	IF NOT fbAdsReadLatchStatus.BUSY THEN
		IF fbAdsReadLatchStatus.ERR THEN
			Error := TRUE;
			ErrorID := fbAdsReadLatchStatus.ERRID;
		ELSE
			IF iTriggerInput.Edge = FallingEdge THEN
				TouchProbeActive[iTriggerInput.TouchProbe] := stTouchProbeStatusResponse.FallingEdgeActive;
				TouchProbeValid[iTriggerInput.TouchProbe] := stTouchProbeStatusResponse.FallingEdgeValid;
				TouchProbeValue[iTriggerInput.TouchProbe] := stTouchProbeStatusResponse.FallingEdgeValue;
				TouchProbeCounter[iTriggerInput.TouchProbe] := stTouchProbeStatusResponse.FallingEdgeCounter;
			ELSE
				TouchProbeActive[iTriggerInput.TouchProbe] := stTouchProbeStatusResponse.RisingEdgeActive;
				TouchProbeValid[iTriggerInput.TouchProbe] := stTouchProbeStatusResponse.RisingEdgeValid;
				TouchProbeValue[iTriggerInput.TouchProbe] := stTouchProbeStatusResponse.RisingEdgeValue;
				TouchProbeCounter[iTriggerInput.TouchProbe] := stTouchProbeStatusResponse.RisingEdgeCounter;
			END_IF
			IF TouchProbeValid[iTriggerInput.TouchProbe] = 1 THEN
				IF  iTriggerInput.Mode <> TOUCHPROBEMODE_CONTINOUS		(* single mode *)
					OR LastTouchProbeValue[ iTriggerInput.TouchProbe ] <> TouchProbeValue[ iTriggerInput.TouchProbe ] 	(* or continous mode and value changed *)
					OR LastTouchProbeCounter[ iTriggerInput.TouchProbe ] <> TouchProbeCounter[ iTriggerInput.TouchProbe ](* or continous mode and counter changed *)
					THEN (* new position recorded  *)
					RecordedPosition:=TouchProbeValue[iTriggerInput.TouchProbe];
					LastTouchProbeValue := TouchProbeValue;
					LastTouchProbeCounter := TouchProbeCounter;
					Done := TRUE;
					IF TriggerInput.ModuloPositions AND (ModuloFactor<>0) THEN	(* check for  (ModuloFactor=0) - 2007-02-06 KSt *)
						RecordedPosition := MODABS(RecordedPosition,  ModuloFactor);
						TouchProbeModuloValue[TriggerInput.TouchProbe] := RecordedPosition;
(*						InWindow := (RecordedPosition>=FirstPosition) AND (RecordedPosition<=LastPosition);*)	(* 20110216 KSt *)
						IF FirstPosition>LastPosition THEN (* 20110216 KSt *)
							InWindow := (RecordedPosition>=FirstPosition) OR  (RecordedPosition<=LastPosition);  (* 20110216 KSt *)
						ELSE
							InWindow := (RecordedPosition>=FirstPosition) AND (RecordedPosition<=LastPosition);
						END_IF
					ELSE
						InWindow := (RecordedPosition>=FirstPosition) AND (RecordedPosition<=LastPosition);
					END_IF
					IF WindowOnly AND NOT InWindow THEN
						RecordedPosition:=0;
						Done := FALSE;
						Restart := TRUE; (* ignore this event, latch next one *)
					ELSE
						(* fill RecordedData structure *)
						RecordedData.RecordedPosition := RecordedPosition;
						RecordedData.Counter:=TouchProbeCounter[TriggerInput.TouchProbe];
						RecordedData.AbsolutePosition := TouchProbeValue[iTriggerInput.TouchProbe];
						IF ModuloFactor = 0 THEN
							RecordedData.ModuloPosition := MODABS(RecordedData.AbsolutePosition,  360);
						ELSE
							RecordedData.ModuloPosition := MODABS(RecordedData.AbsolutePosition,  ModuloFactor);
						END_IF
					END_IF
					iState := STATE_INITIALIZATION;
				END_IF
			ELSIF TouchProbeActive[iTriggerInput.TouchProbe] <> 1 THEN
				TouchProbeInactiveCounter[iTriggerInput.TouchProbe] := TouchProbeInactiveCounter[iTriggerInput.TouchProbe] + 1;
				IF TouchProbeInactiveCounter[iTriggerInput.TouchProbe] > 1 THEN
					(* error condition when the probing sequence is inactive more than once *)
					Error := TRUE;
					ErrorID := MC_ERROR_TOUCH_PROBE_DEACTIVATED;
					CommandAborted := TRUE;
					iState := STATE_INITIALIZATION;
				END_IF
			END_IF
		END_IF
		fbAdsReadLatchStatus(WRTRD:=FALSE); (* reset *)
		IF iTriggerInput.Mode=TOUCHPROBEMODE_CONTINOUS AND Execute THEN
			fbAdsReadLatchStatus(WRTRD:=TRUE); (* retrigger *)
		END_IF
	END_IF
END_IF
END_ACTION

ACTION ActTouchProbeMonitorLatchValid:
(* monitor if the touch probe has been triggered *)

IF F_AxisExternalLatchValid(Axis.NcToPlc.StateDWord) THEN
	(* read the status of the latch *)
	fbAdsReadValid(	NETID:= TcMcGlobal.NCNETID_TCMC,
				PORT:=AMSPORT_R0_NCSAF ,
				IDXGRP:=16#5100+TriggerInput.EncoderID ,
				IDXOFFS:= 16#202,
				LEN:= SIZEOF(TouchProbeValid[1]),
				DESTADDR:=ADR(TouchProbeValid) ,
				READ:=TRUE ,
				TMOUT:=TcMcGlobal.tADSTimeOut );
	(* read the latched value *)
	fbAdsReadValue(	NETID:= TcMcGlobal.NCNETID_TCMC,
				PORT:=AMSPORT_R0_NCSAF ,
				IDXGRP:=16#5100+TriggerInput.EncoderID ,
				IDXOFFS:= 16#205,
				LEN:=SIZEOF(TouchProbeValue[1]),
				DESTADDR:=ADR(TouchProbeValue) ,
				READ:=TRUE ,
				TMOUT:=TcMcGlobal.tADSTimeOut );
	IF NOT fbAdsReadValid.BUSY AND NOT fbAdsReadValue.BUSY THEN
		IF fbAdsReadValid.err THEN
			Error := TRUE;
			ErrorID := fbAdsReadValid.ERRID;
			iState := STATE_INITIALIZATION;
		ELSIF fbAdsReadValue.err THEN
			Error := TRUE;
			ErrorID := fbAdsReadValue.ERRID;
			iState := STATE_INITIALIZATION;
		ELSE (* no error *)
			IF TouchProbeValid[TriggerInput.TouchProbe]=1 THEN
				RecordedPosition:=TouchProbeValue[TriggerInput.TouchProbe];
				Done := TRUE;
//				IF TriggerInput.ModuloPositions AND (ModuloFactor<>0) THEN	(* check for  (ModuloFactor=0) - 2007-02-06 KSt *)
				IF TriggerInput.ModuloPositions THEN	(* check for  (ModuloFactor=0) - 2007-02-06 KSt *)
//					RecordedPosition := MODABS(RecordedPosition,  ModuloFactor);
					IF ModuloFactor = 0 THEN (* not supposed to happen here - 2017-04-28 KSt *)
						RecordedPosition := MODABS(RecordedPosition,  360); (* default 360 not supposed to happen here - 2017-04-28 KSt *)
					ELSE
						RecordedPosition := MODABS(RecordedPosition,  ModuloFactor);
					END_IF
					TouchProbeModuloValue[TriggerInput.TouchProbe] := RecordedPosition;
(*					InWindow := (RecordedPosition>=FirstPosition) AND (RecordedPosition<=LastPosition);*)  (* 20110216 KSt *)
					IF FirstPosition>LastPosition THEN (* 20110216 KSt *)
						InWindow := (RecordedPosition>=FirstPosition) OR  (RecordedPosition<=LastPosition);  (* 20110216 KSt *)
					ELSE
						InWindow := (RecordedPosition>=FirstPosition) AND (RecordedPosition<=LastPosition);
					END_IF
				ELSE
					InWindow := (RecordedPosition>=FirstPosition) AND (RecordedPosition<=LastPosition);
				END_IF
				IF WindowOnly AND NOT InWindow THEN
					RecordedPosition:=0;
					Done := FALSE;
					Restart := TRUE; (* ignore this event, latch next one *)
				ELSE
					(* fill RecordedData structure *)
					RecordedData.RecordedPosition := RecordedPosition;
					RecordedData.Counter:=TouchProbeCounter[TriggerInput.TouchProbe];
					RecordedData.AbsolutePosition := TouchProbeValue[TriggerInput.TouchProbe];
					IF ModuloFactor = 0 THEN
						RecordedData.ModuloPosition := MODABS(RecordedData.AbsolutePosition,  360);
					ELSE
						RecordedData.ModuloPosition := MODABS(RecordedData.AbsolutePosition,  ModuloFactor);
					END_IF
				END_IF
				iState := STATE_INITIALIZATION;
			ELSE
				fbAdsReadValid(READ:=FALSE);
				fbAdsReadValue(READ:=FALSE);
			END_IF
		END_IF
	END_IF
END_IF
END_ACTION

ACTION ActTouchProbeMonitorPlcEvent:
(* touch probe sequence for simple PLC inputs *)
(* monitor PLC input trigger *)

RtrigPlcEvent(CLK:=TriggerInput.PlcEvent);
FtrigPlcEvent(CLK:=TriggerInput.PlcEvent);
IF ((TriggerInput.Edge=RisingEdge) AND RtrigPlcEvent.Q) OR
   ((TriggerInput.Edge=FallingEdge) AND FtrigPlcEvent.Q) THEN
	RecordedPosition:=Axis.NcToPlc.ActPos; 	(* 2007-02-06 KSt *)
	IF TriggerInput.ModuloPositions AND (ModuloFactor<>0) THEN	(* check for  (ModuloFactor=0) - 2007-02-06 KSt *)
		RecordedPosition :=  MODABS(RecordedPosition,  ModuloFactor);
(*		InWindow := (RecordedPosition>=FirstPosition) AND (RecordedPosition<=LastPosition);*)  (* 20110216 KSt *)
		IF FirstPosition>LastPosition THEN (* 20110216 KSt *)
			InWindow := (RecordedPosition>=FirstPosition) OR  (RecordedPosition<=LastPosition);  (* 20110216 KSt *)
		ELSE
			InWindow := (RecordedPosition>=FirstPosition) AND (RecordedPosition<=LastPosition);
		END_IF
	ELSE
		InWindow := (RecordedPosition>=FirstPosition) AND (RecordedPosition<=LastPosition);
	END_IF
	IF WindowOnly AND NOT InWindow THEN
		RecordedPosition:=0;	(* 2007-02-06 KSt *)
	ELSE
		(* fill RecordedData structure *)
		RecordedData.RecordedPosition := RecordedPosition;
		RecordedData.Counter := RecordedData.Counter + 1;
		RecordedData.AbsolutePosition := Axis.NcToPlc.ActPos;
		IF ModuloFactor = 0 THEN
			RecordedData.ModuloPosition := MODABS(RecordedData.AbsolutePosition,  360);
		ELSE
			RecordedData.ModuloPosition := MODABS(RecordedData.AbsolutePosition,  ModuloFactor);
		END_IF
		Done := TRUE;
		iState := STATE_INITIALIZATION;
	END_IF
END_IF
END_ACTION

ACTION ActTouchProbeStartupInit:
(* initialization on plc start-up *)
(* read the axis' modulo factor *)

IF TriggerInput.ModuloPositions THEN
	IF ModuloFactor = 0 THEN
		InitDone := FALSE; (* 2007-02-06 KSt *)
	END_IF
	fbAdsReadModulo(	NETID:= TcMcGlobal.NCNETID_TCMC,
						PORT:= AMSPORT_R0_NCSAF,
						IDXGRP:= 16#5000+TriggerInput.EncoderID ,
						IDXOFFS:= 16#9,
						LEN:= SIZEOF(tempModuloFactor), (* ModuloFactor changed to tempModuloFactor - 2017-40-28 KSt *)
						DESTADDR:= ADR(tempModuloFactor),
						READ:= TRUE,
						TMOUT:= TcMcGlobal.tADSTimeOut);
	IF NOT fbAdsReadModulo.BUSY THEN
		IF fbAdsReadModulo.ERR OR (tempModuloFactor=0) THEN
			fbAdsReadModulo( READ:=FALSE ); 	(* 2007-02-06 KSt *)
			InitDone := FALSE; 	(* init failed - 2007-02-06 KSt *)
			Error := TRUE;
			ErrorID := fbAdsReadModulo.ERRID;
		ELSE
			ModuloFactor := tempModuloFactor; (* take as valid ModuloFactor - 2017-04-28 KSt *) 
			InitDone := TRUE;
		END_IF
	END_IF
ELSE (* no modulo positions *)
	fbAdsReadModulo( READ:=FALSE );	(* 2007-02-06 KSt *)
	InitDone := TRUE;
END_IF
END_ACTION

END_FUNCTION_BLOCK

// POUs/Administrative/Touch Probe/MC_AbortTrigger
FUNCTION_BLOCK MC_AbortTrigger
(*	The function block is used to abort function blocks which are connected to
	trigger events (e.g. MC_TouchProbe) 
*)
VAR_IN_OUT
	Axis			:	AXIS_REF; (*Reference to an axis*)
	TriggerInput	: 	TRIGGER_REF; 		(* Reference to the trigger signal source. *)
END_VAR
VAR_INPUT
	Execute		:	BOOL;		(* Starts aborting  touch probe sequence *)
END_VAR
VAR_OUTPUT
	Done		:	BOOL;		(* function completed *)
	Busy		: 	BOOL;		(* function block is currently Busy *)
	Error		:	BOOL;		(* Signals that error has occurred within Function Block *)
{attribute 'displaymode':='hex'}
	ErrorID		:	UDINT;		(* Error identification *)
END_VAR
VAR
	ADSbusy	: 	BOOL;
	fbADSwrite	: 	ADSWRITE;
	i: INT;
	iState		: 	_E_TcMC_STATES := STATE_INITIALIZATION;
END_VAR
VAR
	LatchID		: 	UDINT;
	fbOnTrigger	: 	R_TRIG;
	stTouchProbeDeactivation : _ST_TcNc_TouchProbeDeactivation;
END_VAR

IF NOT Execute THEN
	Done := FALSE;
	Error := FALSE;			(* reset at falling edge of Execute *)
	ErrorID := 0;
END_IF

fbOnTrigger(CLK:= Execute);

FOR i := 1 TO 2 DO (* typically aborted after one scan *)
	CASE iState OF
		STATE_INITIALIZATION :

			IF fbOnTrigger.Q OR fbADSwrite.BUSY THEN
				Busy := TRUE;

				IF fbOnTrigger.Q THEN
					(* initialization *)
					Done := FALSE;
					Error := FALSE;
					ErrorID := 0;
					fbADSwrite(WRITE:=FALSE);
					IF TriggerInput.EncoderID > 255 THEN
						Error := TRUE;
						ErrorID := MC_ERROR_INVALID_TOUCH_PROBE;
					END_IF
				END_IF

				IF TcMcGlobal.NcDeviceInfoNcVersion=0 THEN
					(* read version of NC *)
					TcMcGlobal.ReadDeviceInfo();
					iState := STATE_WAITING;
					EXIT; (* FOR loop *)
				ELSIF NOT Error THEN
					iState := STATE_ORDER;
				END_IF
			END_IF

		STATE_WAITING :	(* 2013-09-04 - new waiting state in case of invalid NC version information *)
			(* check for NC version *)
			TcMcGlobal.ReadDeviceInfo();
			IF NOT TcMcGlobal.fbADSRDDEVINFO.BUSY THEN
				istate := STATE_ORDER;
			ELSE
				EXIT; (* FOR loop *)
			END_IF

		STATE_ORDER :
			CASE TriggerInput.TouchProbe OF
				TouchProbe1,
				TouchProbe2,
				TouchProbe3,
				TouchProbe4:
					IF TcMcGlobal.NcDeviceInfoNcVersion > 16#020B07DD AND (TriggerInput.mode<>TOUCHPROBEMODE_SINGLE_COMPATIBILITYMODE) THEN
						(* new touch probe interface since TwinCAT 2.11 Nc-Driver 2014 *)
						stTouchProbeDeactivation.TouchProbe := TriggerInput.TouchProbe;
						stTouchProbeDeactivation.Edge := TriggerInput.Edge;
						fbADSwrite(	NETID:= TcMcGlobal.NCNETID_TCMC,
									PORT:=AMSPORT_R0_NCSAF ,
									IDXGRP:=16#5200+TriggerInput.EncoderID ,
									IDXOFFS:=16#205,	(* deactivate touch probe *)
									LEN:= SIZEOF(stTouchProbeDeactivation),
									SRCADDR:=ADR(stTouchProbeDeactivation),
									WRITE:=TRUE ,
									TMOUT:=TcMcGlobal.tADSTimeOut);
					ELSE
						(* classic touch probe interface *)
						fbADSwrite(	NETID:= TcMcGlobal.NCNETID_TCMC,
									PORT:=AMSPORT_R0_NCSAF ,
									IDXGRP:=16#5200+TriggerInput.EncoderID ,
									IDXOFFS:=16#205,	(* deactivate touch probe *)
									LEN:= 0,
									SRCADDR:=0,
									WRITE:=TRUE ,
									TMOUT:=TcMcGlobal.tADSTimeOut);
					END_IF
					IF NOT fbADSwrite.BUSY THEN
						Error := fbADSwrite.ERR;
						ErrorID := fbADSwrite.ERRID;
						TriggerInput.ProbeState := SEL(Error, TouchProbeAborted, TriggerInput.ProbeState );
						Done := NOT Error;
						iState := STATE_INITIALIZATION;	(* 2014-03-21 KSt *)
					END_IF

				PlcEvent:
					(* no action necessary here *);
					TriggerInput.ProbeState := TouchProbeAborted;
					Done := TRUE;
					iState := STATE_INITIALIZATION;	(* 2014-03-21 KSt *)

				ELSE (* case *)
					Error := TRUE;
					ErrorID := MC_ERROR_INVALID_TOUCH_PROBE;
					iState := STATE_INITIALIZATION;	(* 2014-03-21 KSt *)
			END_CASE
			EXIT; (* FOR loop *)
END_CASE
END_FOR

ADSbusy := fbAdsWrite.BUSY;
IF iState=STATE_INITIALIZATION THEN
	(* reset Busy immediately  when sequence ends *)
	Busy := FALSE;
END_IF

END_FUNCTION_BLOCK

// POUs/Motion/Gearing/MC_GearInDyn
FUNCTION_BLOCK MC_GearInDyn
(*	MC_GearInDyn couples a slave axis to a master axis
 *	using a floating point gear ratio. The gear ratio can be 
 *	dynamically modified every PLC cycle as long as the 
 *	Execute input is TRUE.
 *	The acceleration input specifies the maximum slave
 *	acceleration in case of high gear ratio changes.
 *)
VAR_IN_OUT
	Master			:	AXIS_REF; (*Reference to an axis*)
	Slave			:	AXIS_REF; (*Reference to an axis*)
END_VAR
VAR_INPUT
	Enable			:	BOOL;
	GearRatio		:	LREAL := 1.0;
	Acceleration		:	LREAL;
	Deceleration		:	LREAL;	(* not used *)
	Jerk				:	LREAL;	(* not used *)
	BufferMode		:	MC_BufferMode;	
	Options			: 	ST_GearInDynOptions;	(* optional parameters *)
END_VAR
VAR_OUTPUT
	InGear				:	BOOL;
	Busy				: 	BOOL;
	Active				: 	BOOL;
	CommandAborted		:	BOOL;
	Error				:	BOOL;
{attribute 'displaymode':='hex'}
	ErrorID				:	UDINT;
END_VAR
VAR
	LastExecutionResult: 	_ST_FunctionBlockResults;
	ADSbusy: BOOL;
	iState			:	_E_TcMC_STATES := STATE_INITIALIZATION;
	iSubState		: 	INT;
	fbAdsWrite		:	ADSWRITE;
	fbAdsRead		:	ADSREAD;
	sCouple			:	_ST_TcNC_CoupleSlave;
	v_max			: 	LREAL;
	pa_limit			: 	LREAL;
	WasInGear: BOOL;
END_VAR
VAR
{attribute 'conditionalshow'}
	iAcceleration		: 	LREAL;
{attribute 'conditionalshow'}
	TimerStateFeedback: TON;
END_VAR

IF NOT (_F_TcMC_IsValidAxisRef(Master) AND _F_TcMC_IsValidAxisRef(Slave)) THEN // AXIS REFERENCE CHECK - 2020-09-17 KSt
	Error := TRUE;
	ErrorID := MC_ERROR_INVALIDREFERENCE;
	RETURN;
END_IF


CASE iState OF
	STATE_INITIALIZATION:	(* *)
		Busy := FALSE;
		Active := FALSE;
		IF Enable THEN
			Busy := TRUE;
			Active := TRUE;
			fbAdsRead(READ:=FALSE);
			fbAdsWrite(WRITE:=FALSE);
			(* initialize output values *)
			iAcceleration := Acceleration;
			ErrorID := 0;
			Error := FALSE;
			LastExecutionResult.Done := FALSE;
			LastExecutionResult.CommandAborted := FALSE;
			LastExecutionResult.Error := FALSE;
			LastExecutionResult.ErrorID := 0;
			TimerStateFeedback(IN:=FALSE);
			WasInGear := FALSE;
			iSubState := 0;

			IF BufferMode <> 0 THEN
				Error := TRUE;
				ErrorID := MC_ERROR_BUFFERMODE_NOT_SUPPORTED;
			ELSE
				InGear := F_AxisIsCoupled(Slave.NcToPlc.CoupleState) ;
				istate := SEL( InGear, STATE_ORDER, STATE_RUNNING);
			END_IF
		ELSE
			Error := FALSE;	(* reset at falling edge of Execute *)
			ErrorID := 0;
			CommandAborted := FALSE;
			InGear := FALSE;
		END_IF

	STATE_ORDER :
		Slave.PlcToNc.AxisModeLReal := GearRatio; (* 2008-06-02 KSt *)

		CASE iSubState OF
			0 :	(* read maximum master velocity *)
				fbAdsRead(	NETID:= TcMcGlobal.NCNETID_TCMC,
						PORT:= TcMcGlobal.NCPORT_TCMC,
						IDXGRP:=TcMcGlobal.Axis.Parameter.IDXGRP+Master.NcToPlc.AxisId,
						IDXOFFS:= TcMcGlobal.Axis.Parameter.IDXOFFS.VELOMAXIMUM,
						LEN:= SIZEOF(v_max),
						DESTADDR:= ADR(v_max),
						READ:= TRUE,
						TMOUT:= TcMcGlobal.tADSTimeOut);
				IF NOT fbAdsRead.Busy THEN
					Error := fbAdsRead.ERR;
					ErrorID := fbAdsRead.ERRID;
					fbAdsRead(READ:=FALSE);
					IF Error THEN
						iState := STATE_INITIALIZATION;
					ELSE
						iSubState := SEL(iAcceleration=0, iSubState + 2, iSubState + 1 );
					END_IF
				END_IF;

			1 :	(* read slave default acceleration *)
				fbAdsRead(	NETID:=TcMcGlobal.NCNETID_TCMC,
						PORT:= TcMcGlobal.NCPORT_TCMC,
						IDXGRP:=TcMcGlobal.Axis.Parameter.IDXGRP+Slave.NcToPlc.AxisId,
						IDXOFFS:= TcMcGlobal.Axis.Parameter.IDXOFFS.ACC,
						LEN:= SIZEOF(iAcceleration),
						DESTADDR:= ADR(iAcceleration),
						READ:= TRUE,
						TMOUT:= TcMcGlobal.tADSTimeOut);
				IF NOT fbAdsRead.Busy THEN
					Error := fbAdsRead.ERR;
					ErrorID := fbAdsRead.ERRID;
					fbAdsRead(READ:=FALSE);
					IF Error THEN
						iState := STATE_INITIALIZATION;
					ELSE
						iSubState := iSubState + 1;
					END_IF
				END_IF;

			2 : (* couple with dynamic gear ratio *)
				(* 	pa entspricht indirekt, naemlich bezogen auf eine maximale
					Mastergeschwindigkeit, einer maximal erlaubten 
					Beschleunigung (pa = aSlaveMax / vMasterMax ). 
					Der Begrenzungsparameter pa entspricht dabei dem 
					Kehrwert der Hochlaufzeit tH = 1 / pa . 
				*)
				IF iAcceleration > 0 AND v_max > 0 THEN
					pa_limit := iAcceleration / v_max;
				ELSE
					pa_limit := 1;
				END_IF

				sCouple.nSlaveType 	:= INT_TO_UDINT( SEL( Options.CCVmode,
					TCNC_SLAVETYPE_LINEAR_CYCLICCHANGES_RAMP,
					TCNC_SLAVETYPE_CONST_SURFACEVELO_RAMP) );
				sCouple.nMasterAxisId	:= Master.NcToPlc.AxisId;
				sCouple.nMasterSubIdx	:= 0;
				sCouple.nSlaveSubIdx		:= 0;
				sCouple.fCoupleParam1	:= pa_limit;
				sCouple.fCoupleParam2	:= 0;(* unused *)
				sCouple.fCoupleParam3	:= 0;(* unused *)
				sCouple.fCoupleParam4	:= 0;(* unused *)

				(* Slave.PlcToNc.AxisModeLReal := GearRatio;*) (* 2008-06-02 KSt *)

				fbAdsWrite(	NETID:= TcMcGlobal.NCNETID_TCMC,
						PORT:= TcMcGlobal.NCPORT_TCMC_COUPLING,
						IDXGRP:=TcMcGlobal.Axis.Functions.IDXGRP+Slave.NcToPlc.AxisId,
						IDXOFFS:= TcMcGlobal.Axis.Functions.IDXOFFS.CPL,
						LEN:= SIZEOF(sCouple),
						SRCADDR:= ADR(sCouple),
						WRITE:= TRUE,
						TMOUT:= TcMcGlobal.tADSTimeOut);
				IF NOT fbAdsWrite.Busy THEN
					Error := fbAdsWrite.ERR;
					ErrorID := fbAdsWrite.ERRID;
					fbAdsWrite(WRITE:=FALSE);
					IF Error THEN
						iState := STATE_INITIALIZATION;
					ELSE
						InGear := F_AxisIsCoupled(Slave.NcToPlc.CoupleState);
						iState := STATE_RUNNING;
					END_IF
				END_IF
		END_CASE

	STATE_RUNNING:  (* cyclic change of the gear ratio until decoupled or until Execute=FALSE *)
		TimerStateFeedback(IN:=TRUE, PT:=t#50ms); (* 5.7.2006 KSt *)
		Slave.PlcToNc.AxisModeLReal := GearRatio;
		InGear := F_AxisIsCoupled(Slave.NcToPlc.CoupleState) ;
		IF InGear THEN
			WasInGear := TRUE; (* feedback seen, 5.7.2006 KSt *)
		END_IF
		IF (NOT Enable OR NOT InGear) AND (WasInGear OR TimerStateFeedback.Q) THEN (* 5.7.2006 KSt *)
			(* Slave.PlcToNc.AxisModeLReal := 0;*) (* stop when still in gear but not enabled *) (* keep latest gear ratio - 2009-02-19 KSt *)
			CommandAborted := NOT InGear;
			iState := STATE_INITIALIZATION;
		END_IF;

	ELSE  (* CASE : Unknown program state *)
		Error := TRUE;
		ErrorID := 16#FFFFFFFF;
		iState:= STATE_INITIALIZATION;
END_CASE

ADSbusy := fbAdsWrite.BUSY OR fbAdsRead.BUSY;
IF iState=STATE_INITIALIZATION THEN
	(* reset Busy immediately  when sequence ends *)
	IF Busy THEN
		LastExecutionResult.Done := InGear;
		LastExecutionResult.CommandAborted := CommandAborted;
		LastExecutionResult.Error := Error;
		LastExecutionResult.ErrorID := ErrorID;
	END_IF
	Busy := FALSE;
	Active := FALSE;
END_IF

END_FUNCTION_BLOCK

// POUs/Administrative/Extensions/MC_PowerStepper
FUNCTION_BLOCK MC_PowerStepper
VAR_IN_OUT
	Axis		:	AXIS_REF; (*Reference to an axis*)
END_VAR
VAR_INPUT
	Enable			:	BOOL;
	Enable_Positive	:	BOOL;
	Enable_Negative	:	BOOL;
	Override			:	LREAL := 100.0; (* in percent *)
	DestallParams	:	ST_PowerStepperStruct;
	KL_Status		:	USINT;
	KL_Status2		:	UINT;
END_VAR
VAR_OUTPUT
	Status			:	BOOL;
	Error			:	BOOL;
{attribute 'displaymode':='hex'}
	ErrorID			:	UDINT;
	Stalled			:	BOOL;
	StallError			:	BOOL;
END_VAR
VAR
	fbPower			:	MC_Power;
	ErrorCode		:	DWORD;
	fbWriteErrCode	:	ADSWRITE;
	nRefState		:	DWORD;
	fbWriteNonRef	:	ADSWRITE;
	fbReadParams	:	ADSREAD;
	fbWriteInstOvr		:	ADSWRITE;
	bAdsInitDone		:	BOOL;

	bOverTemp		:	BOOL;
	rtOverTemp		:	R_TRIG;
	bUnderVoltage	:	BOOL;
	rtUnderVoltage	:	R_TRIG;
	bOpenLoopA		:	BOOL;
	rtOpenLoopA		:	R_TRIG;
	bOpenLoopB		:	BOOL;
	rtOpenLoopB		:	R_TRIG;
	bOverCurrentA	:	BOOL;
	rtOverCurrentA	:	R_TRIG;
	bOverCurrentB	:	BOOL;
	rtOverCurrentB	:	R_TRIG;
	rtStallError		:	R_TRIG;
	bOldState		:	BOOL;

	bLagFilterInit		: 	BOOL;
	tonLagFilter		:	TON;
	tonNoLagFilter	:	TON;

	wState2			:	WORD;
	nAngle			:	INT;
	nOldAngle		:	INT;
	AngleDiff			:	INT;
	bInErrorState		:	BOOL;

	nParamIdx		:	INT;
	bParamEnabled	:	BOOL;
	fLagLimit			:	LREAL;
	fLagFilter			:	LREAL;
	nTries			:	INT;
	tTimeOut			:	TON;
END_VAR

(*
	Aufruf des Standard-Bausteins
*)
fbPower(
	Enable:=Enable,
	Enable_Positive:=Enable_Positive,
	Enable_Negative:=Enable_Negative,
	Override:=Override,
	Axis:=Axis);

(*
	Ein paar Vorbereitungen ...
*)
wState2:=UINT_TO_WORD(KL_Status2);
bInErrorState:=Axis.NcToPlc.ErrorCode<>0;
nAngle:=SHR(USINT_TO_BYTE(KL_Status),1) AND 7;
AngleDiff:=nAngle-nOldAngle;
nOldAngle:=nAngle;
IF((Axis.NcToPlc.StateDWord AND 16#0000001C)=16#0000001C)THEN		(* Ziel erreicht *)
	nTries:=0;
END_IF
IF((Axis.NcToPlc.StateDWord AND 16#00000080)=16#00000080)THEN		(* Stop *)
	nTries:=0;
END_IF

(* ======================================
	Parameter-Lademaschine
====================================== *)
IF(NOT Enable)THEN
	(*
		Reinitialisieren
	*)
	nParamIdx:=0;
	bParamEnabled:=FALSE;
	fbReadParams(
		NETID:='', PORT:=AMSPORT_R0_NCSAF, IDXGRP:=0, IDXOFFS:=0,
		LEN:=0, DESTADDR:=0,
		READ:=FALSE, TMOUT:=T#5s);
ELSE
	IF(NOT bParamEnabled)THEN
		CASE nParamIdx OF
			0:
				IF(NOT fbReadParams.READ)THEN
					fbReadParams.LEN:=SIZEOF(fLagLimit);
					fbReadParams.DESTADDR:=ADR(fLagLimit);
					fbReadParams.IDXGRP:=16#00004000+Axis.NcToPlc.AxisId;
					fbReadParams.IDXOFFS:=16#00020012;
					fbReadParams.READ:=TRUE;
				ELSIF(NOT fbReadParams.BUSY)THEN
					IF(fbReadParams.ERR)THEN
						fLagLimit:=5.0;
					END_IF
					fbReadParams.READ:=FALSE;
					nParamIdx:=nParamIdx+1;
				END_IF
				fbReadParams(NETID:='', PORT:=AMSPORT_R0_NCSAF, TMOUT:=T#5s);
			1:
				IF(NOT fbReadParams.READ)THEN
					fbReadParams.LEN:=SIZEOF(fLagFilter);
					fbReadParams.DESTADDR:=ADR(fLagFilter);
					fbReadParams.IDXGRP:=16#00004000+Axis.NcToPlc.AxisId;
					fbReadParams.IDXOFFS:=16#00020013;
					fbReadParams.READ:=TRUE;
				ELSIF(NOT fbReadParams.BUSY)THEN
					IF(fbReadParams.ERR)THEN
						fLagFilter:=0.1;
					END_IF
					fbReadParams.READ:=FALSE;
					nParamIdx:=nParamIdx+1;
					tonLagFilter(IN:=FALSE, PT:=T#10ms);
					tonNoLagFilter(IN:=NOT tonLagFilter.IN, PT:=T#10ms);
				END_IF
				fbReadParams(NETID:='', PORT:=AMSPORT_R0_NCSAF, TMOUT:=T#5s);
			ELSE
				bParamEnabled:=TRUE;
		END_CASE
	END_IF
END_IF

IF(fbPower.Error)THEN
	ErrorID := fbPower.ErrorID;
	Error := TRUE;
	Status := bAdsInitDone := FALSE;
ELSIF(NOT Enable)THEN
	ErrorID := 0;
	Error := Status := bAdsInitDone := FALSE;
ELSE
	(*
		Sicherstellen, dass die ADS-FBs initialisiert sind
	*)
	IF(NOT bAdsInitDone)THEN
		bAdsInitDone := TRUE;
		fbWriteNonRef(
			WRITE:=FALSE,
			NETID:='',
			PORT:=AMSPORT_R0_NCSAF,
			IDXGRP:=16#00004200+Axis.NcToPlc.AxisId,
			IDXOFFS:=16#0000001B,
			LEN:=SIZEOF(nRefState),
			SRCADDR:=ADR(nRefState),
			TMOUT:=T#5s,
			);
		fbWriteInstOvr(
			WRITE:=FALSE,
			NETID:='',
			PORT:=AMSPORT_R0_NCSAF,
			IDXGRP:=16#00004200+Axis.NcToPlc.AxisId,
			IDXOFFS:=16#00000029,
			LEN:=0,
			SRCADDR:=0,
			TMOUT:=T#5s,
			);
		fbWriteErrCode(
			WRITE:=FALSE,
			NETID:='',
			PORT:=AMSPORT_R0_NCSAF,
			IDXGRP:=16#00004200+Axis.NcToPlc.AxisId,
			IDXOFFS:=16#00000019,
			LEN:=SIZEOF(ErrorCode),
			SRCADDR:=ADR(ErrorCode),
			TMOUT:=T#5s,
			);
	END_IF

	(*
		Zentrales Versenden für Kommandos zur instantanen Override-Änderung
		Dies muss vor der Stelle des Test liegen, damit der Override-Wert im Mapping sicher angekommen ist,
		wenn dieses Kommando per ADS eintrifft.
	*)
	fbWriteInstOvr(
		NETID:='',
		PORT:=AMSPORT_R0_NCSAF,
		IDXGRP:=16#00004200+Axis.NcToPlc.AxisId,
		IDXOFFS:=16#00000029,
		LEN:=0,
		SRCADDR:=0,
		TMOUT:=T#5s,
		);
	IF(NOT fbWriteInstOvr.BUSY)THEN
		fbWriteInstOvr.WRITE:=FALSE;
	END_IF

	bLagFilterInit:=bLagFilterInit OR tonLagFilter.Q;

	IF(DestallParams.DestallEnable)THEN
		(*
			Stall Detection
		*)
		bOldState:=Stalled;
		CASE DestallParams.DestallDetectMode OF
			PwStDetectMode_Encoderless:
				Stalled:=ABS(AngleDiff)>=4;
			PwStDetectMode_Lagging:
				IF(bParamEnabled)THEN
					IF(fLagFilter<=0.001)THEN
						tonLagFilter(IN:=FALSE, PT:=T#10ms);
						tonNoLagFilter(IN:=NOT tonLagFilter.IN, PT:=T#10ms);
						Stalled:=ABS(Axis.NcToPlc.PosDiff)>=fLagLimit;
					ELSE
						tonLagFilter(IN:=(ABS(Axis.NcToPlc.PosDiff)>=fLagLimit), PT:=LREAL_TO_TIME(fLagFilter*1000.0));
						tonNoLagFilter(IN:=NOT tonLagFilter.IN, PT:=LREAL_TO_TIME(fLagFilter*1000.0));
						Stalled:=tonLagFilter.Q;
					END_IF
				ELSE
					tonLagFilter(IN:=FALSE, PT:=T#10ms);
					tonNoLagFilter(IN:=NOT tonLagFilter.IN, PT:=T#10ms);
					Stalled:=FALSE;
				END_IF
			ELSE
				Stalled:=FALSE;
		END_CASE
		IF(NOT bOldState AND Stalled)THEN
			nTries:=nTries+1;
		END_IF
		(*
			Stall Handling
		*)
		StallError:=StallError AND (bInErrorState  OR fbWriteErrCode.WRITE);
		bOldState:=StallError;
		CASE DestallParams.DestallMode OF
			PwStMode_None:
				StallError:=FALSE;
				tTimeOut(IN:=FALSE, PT:=T#10ms);
			PwStMode_SetError:
				StallError:=StallError OR Stalled;
				tTimeOut(IN:=FALSE, PT:=T#10ms);
			PwStMode_SetErrNonRef:
				StallError:=StallError OR Stalled;
				IF(Stalled AND ((Axis.NcToPlc.StateDWord AND 16#00000002)<>0) )THEN
					nRefState:=0;
					fbWriteNonRef.WRITE:=TRUE;
				END_IF
				tTimeOut(IN:=FALSE, PT:=T#10ms);
			PwStMode_UseOverride:
				IF(Stalled OR (bLagFilterInit AND NOT tonNoLagFilter.Q))THEN	(* HKP *)
					Axis.PlcToNc.Override := 0;
					fbWriteInstOvr.WRITE:=TRUE;
				END_IF
				tTimeOut(IN:=Stalled, PT:=MAX(DestallParams.Timeout, T#10ms));
				StallError:=StallError OR tTimeOut.Q;
				IF(nTries>DestallParams.Retries)THEN
					StallError:=TRUE;
				END_IF
		END_CASE

		IF(StallError AND NOT bOldState)THEN
			ADSLOGDINT((ADSLOG_MSGTYPE_ERROR OR ADSLOG_MSGTYPE_LOG), 'MC_PowerStepper (AxisID: %d) reporting error 0x4636 (stall error) !', DWORD_TO_DINT(Axis.NcToPlc.AxisId));
		END_IF
		rtStallError(CLK:=StallError AND NOT bInErrorState AND NOT fbWriteErrCode.WRITE);
		IF(rtStallError.Q)THEN
			ErrorCode:=16#00004636;
			fbWriteErrCode.WRITE:=TRUE;
		END_IF

	END_IF

	Status:=TRUE;
	IF(DestallParams.StatusMonEnable)THEN
		(*
			State Monitoring
		*)
		bOldState:=bOverTemp;
		bOverTemp:=(wState2 AND 2#0000000100000000)<>0;
		Status:=Status AND NOT bOverTemp;
		IF(bOverTemp AND NOT bOldState)THEN
			ADSLOGDINT((ADSLOG_MSGTYPE_ERROR OR ADSLOG_MSGTYPE_LOG), 'MC_PowerStepper (AxisID: %d) reporting error 0x4630 (overtemperature, KL terminal) !', DWORD_TO_DINT(Axis.NcToPlc.AxisId));
		END_IF
		rtOverTemp(CLK:=bOverTemp AND NOT bInErrorState AND NOT fbWriteErrCode.WRITE);
		IF(rtOverTemp.Q)THEN
			ErrorCode:=16#00004630;
			fbWriteErrCode.WRITE:=TRUE;
		END_IF
		bOverTemp:=bOverTemp AND (bInErrorState  OR fbWriteErrCode.WRITE);
		bOldState:=bUnderVoltage;
		bUnderVoltage:=(wState2 AND 2#0000001000000000)<>0;
		Status:=Status AND NOT bUnderVoltage;
		IF(bUnderVoltage AND NOT bOldState)THEN
						ADSLOGDINT((ADSLOG_MSGTYPE_ERROR OR ADSLOG_MSGTYPE_LOG), 'MC_PowerStepper (AxisID: %d) reporting error 0x4631 (bad supply voltage, KL terminal) !', DWORD_TO_DINT(Axis.NcToPlc.AxisId));
		END_IF
		rtUnderVoltage(CLK:=bUnderVoltage AND NOT bInErrorState AND NOT fbWriteErrCode.WRITE);
		IF(rtUnderVoltage.Q)THEN
			ErrorCode:=16#00004631;
			fbWriteErrCode.WRITE:=TRUE;
		END_IF
		bUnderVoltage:=bUnderVoltage AND (bInErrorState  OR fbWriteErrCode.WRITE);
		bOldState:=bOpenLoopA;
		bOpenLoopA:=(wState2 AND 2#0000010000000000)<>0;
		Status:=Status AND NOT bOpenLoopA;
		IF(bOpenLoopA AND NOT bOldState)THEN
			ADSLOGDINT((ADSLOG_MSGTYPE_ERROR OR ADSLOG_MSGTYPE_LOG), 'MC_PowerStepper (AxisID: %d) reporting error 0x4632 (open loop, phase A) !', DWORD_TO_DINT(Axis.NcToPlc.AxisId));
		END_IF
		rtOpenLoopA(CLK:=bOpenLoopA AND NOT bInErrorState AND NOT fbWriteErrCode.WRITE);
		IF(rtOpenLoopA.Q)THEN
			ErrorCode:=16#00004632;
			fbWriteErrCode.WRITE:=TRUE;
		END_IF
		bOpenLoopA:=bOpenLoopA AND (bInErrorState  OR fbWriteErrCode.WRITE);
		bOldState:=bOpenLoopB;
		bOpenLoopB:=(wState2 AND 2#0000100000000000)<>0;
		Status:=Status AND NOT bOpenLoopB;
		IF(bOpenLoopB AND NOT bOldState)THEN
			ADSLOGDINT((ADSLOG_MSGTYPE_ERROR OR ADSLOG_MSGTYPE_LOG), 'MC_PowerStepper (AxisID: %d) reporting error 0x4633 (open loop, phase B) !', DWORD_TO_DINT(Axis.NcToPlc.AxisId));
		END_IF
		rtOpenLoopB(CLK:=bOpenLoopB AND NOT bInErrorState AND NOT fbWriteErrCode.WRITE);
		IF(rtOpenLoopB.Q)THEN
			ErrorCode:=16#00004633;
			fbWriteErrCode.WRITE:=TRUE;
		END_IF
		bOpenLoopB:=bOpenLoopB AND (bInErrorState  OR fbWriteErrCode.WRITE);
		bOldState:=bOverCurrentA;
		bOverCurrentA:=(wState2 AND 2#0001000000000000)<>0;
		Status:=Status AND NOT bOverCurrentA;
		IF(bOverCurrentA AND NOT bOldState)THEN
			ADSLOGDINT((ADSLOG_MSGTYPE_ERROR OR ADSLOG_MSGTYPE_LOG), 'MC_PowerStepper (AxisID: %d) reporting error 0x4634 (overcurrent, phase A) !', DWORD_TO_DINT(Axis.NcToPlc.AxisId));
		END_IF
		rtOverCurrentA(CLK:=bOverCurrentA AND NOT bInErrorState AND NOT fbWriteErrCode.WRITE);
		IF(rtOverCurrentA.Q)THEN
			ErrorCode:=16#00004634;
			fbWriteErrCode.WRITE:=TRUE;
		END_IF
		bOverCurrentA:=bOverCurrentA AND (bInErrorState  OR fbWriteErrCode.WRITE);
		bOldState:=bOverCurrentB;
		bOverCurrentB:=(wState2 AND 2#0010000000000000)<>0;
		Status:=Status AND NOT bOverCurrentB;
		IF(bOverCurrentB AND NOT bOldState)THEN
			ADSLOGDINT((ADSLOG_MSGTYPE_ERROR OR ADSLOG_MSGTYPE_LOG), 'MC_PowerStepper (AxisID: %d) reporting error 0x4635 (overcurrent, phase B) !', DWORD_TO_DINT(Axis.NcToPlc.AxisId));
		END_IF
		rtOverCurrentB(CLK:=bOverCurrentB AND NOT bInErrorState AND NOT fbWriteErrCode.WRITE);
		IF(rtOverCurrentB.Q)THEN
			ErrorCode:=16#00004635;
			fbWriteErrCode.WRITE:=TRUE;
		END_IF
		bOverCurrentB:=bOverCurrentB AND (bInErrorState  OR fbWriteErrCode.WRITE);
	END_IF

	(*
		Zentrale Versendung von Achs-ErrorCodes
	*)
	fbWriteErrCode(
		NETID:='',
		PORT:=AMSPORT_R0_NCSAF,
		IDXGRP:=16#00004200+Axis.NcToPlc.AxisId,
		IDXOFFS:=16#00000019,
		LEN:=SIZEOF(ErrorCode),
		SRCADDR:=ADR(ErrorCode),
		TMOUT:=T#5s,
		);
	IF(bInErrorState)THEN
		fbWriteErrCode.WRITE:=FALSE;
	END_IF

	(*
		Zentrale Versendung von Referenz-Resets
	*)
	fbWriteNonRef(
		NETID:='',
		PORT:=AMSPORT_R0_NCSAF,
		IDXGRP:=16#00004200+Axis.NcToPlc.AxisId,
		IDXOFFS:=16#0000001B,
		LEN:=SIZEOF(nRefState),
		SRCADDR:=ADR(nRefState),
		TMOUT:=T#5s,
		);
	IF(NOT fbWriteNonRef.BUSY)THEN
		fbWriteNonRef.WRITE:=FALSE;
	END_IF

END_IF

END_FUNCTION_BLOCK

// POUs/Administrative/Status and Parameter/MC_ReadParameterSet
FUNCTION_BLOCK  MC_ReadParameterSet
(*	This Function Block returns the complete set of axis parameters *)
VAR_IN_OUT
	Parameter 	: 	ST_AxisParameterSet;
	Axis			:	AXIS_REF; (*Reference to an axis*)
END_VAR
VAR_INPUT
	Execute		: 	BOOL;
END_VAR
VAR_OUTPUT
	Done 		: 	BOOL;
	Busy		: 	BOOL;
	Error 		: 	BOOL;
{attribute 'displaymode':='hex'}
	ErrorID 		: 	UDINT;
END_VAR
VAR
	TriggerExecute: R_TRIG;
	state: _E_TcMC_STATES := STATE_INITIALIZATION;
	fbAdsRead		: 	ADSREAD;
	SizeofPayloadData : UDINT;
	SizeofPayloadData64 : ULINT;
END_VAR

TriggerExecute(CLK:=Execute);

CASE state OF
	STATE_INITIALIZATION:
		IF NOT Execute THEN
			Done := FALSE;
			Error := FALSE;	(* reset at falling edge of Execute *)
			ErrorID := 0;
		END_IF
		IF TriggerExecute.Q THEN
			Done := FALSE;
			Busy := TRUE;
			Error := FALSE;
			ErrorID := 0;
			fbAdsRead(READ:=FALSE);
			IF TcMcGlobal.NcDeviceInfoNcVersion=0 THEN
				TcMcGlobal.ReadDeviceInfo();
				state := STATE_WAITING;
			ELSE
				state := STATE_ORDER;
			END_IF
		END_IF

	STATE_WAITING :
		(* check for NC version *)
		TcMcGlobal.ReadDeviceInfo();
		IF TcMcGlobal.NcDeviceInfoNcVersion<>0 THEN
			state := STATE_ORDER;
		ELSIF TcMcGlobal.fbADSRDDEVINFO.ERR THEN
			Error := TRUE;
			ErrorID := TcMcGlobal.fbADSRDDEVINFO.ERRID;
			Busy := FALSE;
			state := STATE_INITIALIZATION;
		END_IF

	STATE_ORDER :
		ActGetSizeOfParameterSet();		(* 2011-06-29 KSt - get size for differently aligned systems *)
		fbAdsRead(
			NETID:= TcMcGlobal.NCNETID_TCMC,
			PORT:= TcMcGlobal.NCPORT_TCMC,
			IDXGRP:=TcMcGlobal.Axis.Parameter.IDXGRP+Axis.NcToPlc.AxisId,
			IDXOFFS:= (* 16#00 + *) Axis.NcToPlc.ControlLoopIndex * 16#00100000,
(*			LEN:= SIZEOF(Parameter),*)	(* 2011-06-29 KSt - get size for differently aligned systems *)
			LEN:= ,						(* 2011-06-29 KSt - get size for differently aligned systems *)
			DESTADDR:= ADR(Parameter),
			READ:= TRUE,
			TMOUT:= TcMcGlobal.tADSTimeOut );
		IF NOT fbAdsRead.BUSY THEN
			Error := fbAdsRead.ERR;
			ErrorID := fbAdsRead.ERRID;
			Done := NOT Error;
			Busy := FALSE;
			state := STATE_INITIALIZATION;
		END_IF

END_CASE

ACTION ActGetSizeOfParameterSet:

(* adjustment of the data size to different system with different alignement *)

SizeofPayloadData64 := ADR(Parameter.arrReserved) - ADR(Parameter);
SizeofPayloadData := ULINT_TO_UDINT(SizeofPayloadData64);

IF SIZEOF(Parameter) < (1024 + 512) / 2 THEN
	(* TC2 environment
	 	set the size of the data structure to 512 if the payload data size (data without reserved bytes) is smaller,
		Otherwise set the size to the size of the payload data.
	*)
	IF TcMcGlobal.NcDeviceInfoNcVersion >= 16#020B049C THEN	(* from 2.11 NC 1180 *)
		fbAdsRead.LEN := MAX( SizeofPayloadData, 512 );
	ELSE
		(* use 512 for any older system with smaller structure definition *)
		fbAdsRead.LEN := 512;
	END_IF
ELSE
	(* TC3 environment with extended size
		set the size of the data structure to 1024 if the payload data size (data without reserved bytes) is smaller,
		Otherwise set the size to the size of the payload data.
	*)
	fbAdsRead.LEN := MAX( SizeofPayloadData, 1024 );
END_IF
END_ACTION

END_FUNCTION_BLOCK

// POUs/Administrative/Status and Parameter/MC_ReadAxisComponents
FUNCTION_BLOCK  MC_ReadAxisComponents
VAR_IN_OUT
	AxisComponents 	: 	ST_AxisComponents;
	Axis				:	AXIS_REF; (*Reference to an axis*)
END_VAR
VAR_INPUT
	Execute: BOOL;
END_VAR
VAR_OUTPUT
	Done : BOOL;
	Busy: BOOL;
	Error : BOOL;
{attribute 'displaymode':='hex'}
	ErrorID : UDINT;
END_VAR
VAR
	TriggerExecute: R_TRIG;
	state: _E_TcMC_STATES := STATE_INITIALIZATION;
	fbAdsRead		: 	ADSREAD;
END_VAR

TriggerExecute(CLK:=Execute);

CASE state OF
	STATE_INITIALIZATION:
		IF NOT Execute THEN
			Done := FALSE;
			Error := FALSE;	(* reset at falling edge of Execute *)
			ErrorID := 0;
		END_IF
		IF TriggerExecute.Q THEN
			Done := FALSE;
			Busy := TRUE;
			Error := FALSE;
			ErrorID := 0;
			fbAdsRead(READ:=FALSE);
		END_IF
		IF Busy THEN
			fbAdsRead(
				NETID:= TcMcGlobal.NCNETID_TCMC,
				PORT:= TcMcGlobal.NCPORT_TCMC,
				IDXGRP:=TcMcGlobal.Axis.Parameter.IDXGRP+Axis.NcToPlc.AxisId,
				IDXOFFS:= 16#5A,
				LEN:= SIZEOF(AxisComponents),
				DESTADDR:= ADR(AxisComponents),
				READ:= TRUE,
				TMOUT:= TcMcGlobal.tADSTimeOut );
			IF NOT fbAdsRead.BUSY THEN
				Error := fbAdsRead.ERR;
				ErrorID := fbAdsRead.ERRID;
				Done := NOT Error;
				Busy := FALSE;
			END_IF
		END_IF
END_CASE

END_FUNCTION_BLOCK

// POUs/Motion/Gearing/MC_GearIn
FUNCTION_BLOCK MC_GearIn
(*	This Function Block commands a ratio between the velocity of the slave and master axis. *)
VAR_IN_OUT
	Master			:	AXIS_REF; (*Reference to an axis*)
	Slave			:	AXIS_REF; (*Reference to an axis*)
END_VAR
VAR_INPUT
	Execute			:	BOOL;			
(*	ContinuousUpdate :	BOOL; *)			(* not available *)
	RatioNumerator	:	LREAL				:= 1; (* changed from INT (PLCopen) to LREAL *)
	RatioDenominator	:	UINT			:= 1;
(*	MasterValueSource :	MC_SOURCE; *)		(* not available *)
	Acceleration		:	LREAL;		
	Deceleration		:	LREAL;		
	Jerk				:	LREAL;		
	BufferMode		:	MC_BufferMode;	
	Options			: 	ST_GearInOptions;	(* optional parameters *)
END_VAR
VAR_OUTPUT
	InGear			:	BOOL;	
	Busy			: 	BOOL;	
	Active			: 	BOOL;	
	CommandAborted	:	BOOL;	
	Error			:	BOOL;	
{attribute 'displaymode':='hex'}
	ErrorID			:	UDINT;	
END_VAR
VAR
	LastExecutionResult	: 	_ST_FunctionBlockResults;
	ADSbusy: BOOL;
	iState				:	_E_TcMC_STATES := STATE_INITIALIZATION;
	fbAdsWrite			:	ADSWRITE;
	sCouple				:	_ST_TcNC_CoupleSlave;
	fbOptGearInDyn		: 	MC_GearInDyn;
END_VAR
VAR
{attribute 'conditionalshow'}
	fbOnTrigger			:	R_TRIG;
{attribute 'conditionalshow'}
	TimerStateFeedback	: 	TON;
END_VAR

IF NOT (_F_TcMC_IsValidAxisRef(Master) AND _F_TcMC_IsValidAxisRef(Slave)) THEN // AXIS REFERENCE CHECK - 2020-09-17 KSt
	Error := TRUE;
	ErrorID := MC_ERROR_INVALIDREFERENCE;
	RETURN;
END_IF

fbOnTrigger(CLK:= Execute);

CASE iState OF
STATE_INITIALIZATION:	(* *)
	Busy := FALSE;
	IF NOT Execute THEN
		InGear := FALSE;
		CommandAborted := FALSE;
		Error := FALSE;			(* reset at falling edge of Execute *)
		ErrorID := 0;
	END_IF
	IF fbOnTrigger.Q THEN
		Busy := TRUE;
		(* initialize output values *)
		InGear 			:= FALSE;
		CommandAborted	:= FALSE;
		ErrorID := 0;
		Error := FALSE;
		LastExecutionResult.Done := FALSE;
		LastExecutionResult.CommandAborted := FALSE;
		LastExecutionResult.Error := FALSE;
		LastExecutionResult.ErrorID := 0;
		fbOptGearInDyn.Enable := FALSE;
		TimerStateFeedback(IN:=FALSE);

		IF RatioDenominator = 0 THEN
			Error := TRUE;
			ErrorID := MC_ERROR_PARAMETER_NOT_CORRECT;
		ELSIF BufferMode <> 0 THEN
			Error := TRUE;
			ErrorID := MC_ERROR_BUFFERMODE_NOT_SUPPORTED;
		ELSE
			CASE Options.SlaveType OF
				0, TCNC_SLAVETYPE_LINEAR :
					(* linear gear ratio coupling *)
					sCouple.nSlaveType 		:= INT_TO_UDINT(TCNC_SLAVETYPE_LINEAR); (* linear coupling *)
					sCouple.nMasterAxisId		:= Master.NcToPlc.AxisId;
					sCouple.nMasterSubIdx	:= 0;
					sCouple.nSlaveSubIdx		:= 0;
					sCouple.fCoupleParam1	:= RatioNumerator / RatioDenominator;
					sCouple.fCoupleParam2	:= 0;(* unused *)
					sCouple.fCoupleParam3	:= 0;(* unused *)
					sCouple.fCoupleParam4	:= 0;(* unused *)
		
					fbAdsWrite(	NETID:= TcMcGlobal.NCNETID_TCMC,
							PORT:= TcMcGlobal.NCPORT_TCMC_COUPLING,
							IDXGRP:=TcMcGlobal.Axis.Functions.IDXGRP+Slave.NcToPlc.AxisId,
							IDXOFFS:= TcMcGlobal.Axis.Functions.IDXOFFS.CPL,
							LEN:= SIZEOF(sCouple),
							SRCADDR:= ADR(sCouple),
							WRITE:= TRUE,
							TMOUT:= TcMcGlobal.tADSTimeOut);
					iState := STATE_ORDER;

				TCNC_SLAVETYPE_LINEAR_CYCLICCHANGES_RAMP,
				TCNC_SLAVETYPE_CONST_SURFACEVELO_RAMP :
					fbOptGearInDyn.Enable := TRUE;
					fbOptGearInDyn.Options.CCVmode := Options.SlaveType=TCNC_SLAVETYPE_CONST_SURFACEVELO_RAMP;	// set CCV mode, 2023-03 KSt
					ActGearInDyn();
					iState := STATE_ORDER;
			ELSE
				Error := TRUE;	(* Optional mode not supported with this function block *)
				ErrorID := MC_ERROR_PARAMETER_NOT_CORRECT;
			END_CASE
		END_IF;
	END_IF;

STATE_ORDER:
	CASE Options.SlaveType OF
		0, TCNC_SLAVETYPE_LINEAR :
			fbAdsWrite();
			IF NOT fbAdsWrite.Busy THEN
				IF fbAdsWrite.Err THEN
					ErrorID := fbAdsWrite.ErrId;
					Error := TRUE;
					iState := STATE_INITIALIZATION;
				ELSE
					iState := STATE_RUNNING;
				END_IF
				fbAdsWrite(WRITE := FALSE);
			END_IF;

		(* optional modes to couple with dynamically changable gear ratio (just couple) *)
		TCNC_SLAVETYPE_LINEAR_CYCLICCHANGES_RAMP,
		TCNC_SLAVETYPE_CONST_SURFACEVELO_RAMP :
			ActGearInDyn();
			IF fbOptGearInDyn.InGear THEN
				InGear := TRUE;
				fbOptGearInDyn.Enable := FALSE;
				ActGearInDyn();
				iState := STATE_INITIALIZATION;
			ELSIF NOT fbOptGearInDyn.Busy THEN
				CommandAborted := fbOptGearInDyn.CommandAborted;
				Error := fbOptGearInDyn.Error;
				ErrorID := fbOptGearInDyn.ErrorID;
				fbOptGearInDyn.Enable := FALSE;
				iState := STATE_INITIALIZATION;
			END_IF
	ELSE
		Error := TRUE;	(* Optional mode not supported with this function block *)
		ErrorID := MC_ERROR_PARAMETER_NOT_CORRECT;
		iState := STATE_INITIALIZATION;
	END_CASE

STATE_RUNNING:  (* Return *)
	TimerStateFeedback(IN:=TRUE, PT:=t#50ms); (* 21.2.2006 KSt *)
	IF  (Slave.NcToPlc.CoupleState = 2) OR (Slave.NcToPlc.CoupleState = 3) THEN
		(* axis successfully coupled *)
		InGear := TRUE;
		iState := STATE_INITIALIZATION;
	ELSIF TimerStateFeedback.Q THEN
		(* 	nCoupleState does not respond 'coupled' - the reason may be
			a MC_GearOut command which aborted the GearIn command *)
		CommandAborted := TRUE;
		iState := STATE_INITIALIZATION;
	END_IF;

ELSE  (* CASE : Unknown program state *)
	Error := TRUE;
	ErrorID := 16#FFFFFFFF;
	iState:= STATE_INITIALIZATION;
END_CASE

ADSbusy := fbAdsWrite.BUSY;
IF iState=STATE_INITIALIZATION THEN
	(* reset Busy immediately  when sequence ends *)
	IF Busy THEN
		LastExecutionResult.Done := InGear;
		LastExecutionResult.CommandAborted := CommandAborted;
		LastExecutionResult.Error := Error;
		LastExecutionResult.ErrorID := ErrorID;
	END_IF
	Busy := FALSE;
END_IF

Active := Busy;

ACTION ActGearInDyn:
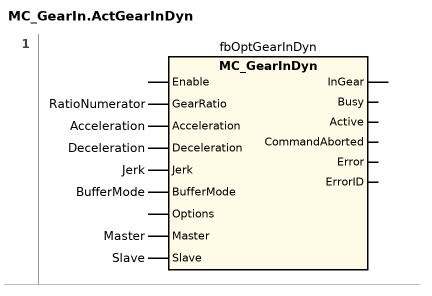
// NETWORK 1
fbOptGearInDyn(
    GearRatio := RatioNumerator,
    Acceleration := Acceleration,
    Deceleration := Deceleration,
    Jerk := Jerk,
    BufferMode := BufferMode,
    Master := Master,
    Slave := Slave); // MC_GearInDyn
END_ACTION

ACTION WriteGearRatio:
	(* action can be called from external in case of coupling modes with dynamically changable gear ratio *)
	IF RatioDenominator = 0 THEN
		Slave.PlcToNc.AxisModeLReal := RatioNumerator;
	ELSE
		Slave.PlcToNc.AxisModeLReal := RatioNumerator / RatioDenominator;
	END_IF
END_ACTION

END_FUNCTION_BLOCK

// POUs/Motion/Gearing/MC_GearOut
FUNCTION_BLOCK MC_GearOut
(*	This Function Block disengages the Slave axis from the Master axis.
	Notes:
	It is assumed that this command is followed by another command, for instance 
	MC_Stop, MC_GearIn, or any other command. If there is no new command, the 
	default condition should be: maintain last velocity.
 *)
VAR_IN_OUT
	Slave			:	AXIS_REF; (*Reference to an axis*)
END_VAR
VAR_INPUT
	Execute			:	BOOL;		
	Options			: 	ST_GearOutOptions;		(* optional parameters *)
END_VAR
VAR_OUTPUT
	Done			:	BOOL;		
	Busy			: 	BOOL;		
	Error			:	BOOL;		
{attribute 'displaymode':='hex'}
	ErrorID			:	UDINT;		
END_VAR
VAR
	LastExecutionResult: 	_ST_FunctionBlockResults;
	ADSbusy		: 	BOOL;
	iState			:	_E_TcMC_STATES := STATE_INITIALIZATION;
	fbAdsWrite		:	ADSWRITE;
END_VAR
VAR
{attribute 'conditionalshow'}
	fbOnTrigger		:	R_TRIG;
{attribute 'conditionalshow'}
	TimerStateFeedback: TON;
END_VAR

IF NOT _F_TcMC_IsValidAxisRef(Slave) THEN // AXIS REFERENCE CHECK - 2020-09-17 KSt
	Error := TRUE;
	ErrorID := MC_ERROR_INVALIDREFERENCE;
	RETURN;
END_IF

fbOnTrigger(CLK:= Execute);

CASE iState OF
	STATE_INITIALIZATION:	(* *)
		Busy := FALSE;
		IF NOT Execute THEN
			Done := FALSE;
			Error := FALSE;			(* reset at falling edge of Execute *)
			ErrorID := 0;
		END_IF
	    	IF fbOnTrigger.Q THEN
			(* initialize output values *)
	    		Busy := TRUE;
			Done := FALSE;
			ErrorID := 0;
			Error := FALSE;
			LastExecutionResult.Done := FALSE;
			LastExecutionResult.CommandAborted := FALSE;
			LastExecutionResult.Error := FALSE;
			LastExecutionResult.ErrorID := 0;
			TimerStateFeedback(IN:=FALSE);
			fbAdsWrite(WRITE := FALSE);

			fbAdsWrite(	NETID:=TcMcGlobal.NCNETID_TCMC,
						PORT:= TcMcGlobal.NCPORT_TCMC_COUPLING, (* 12.7.2006 KSt *)
						IDXGRP:=TcMcGlobal.Axis.Functions.IDXGRP+Slave.NcToPlc.AxisId,
						IDXOFFS:= TcMcGlobal.Axis.Functions.IDXOFFS.DECPL,
						LEN:= 0,
						SRCADDR:= 0,
						WRITE:= TRUE,
						TMOUT:= TcMcGlobal.tADSTimeOut);

			iState := STATE_ORDER;
		END_IF;

	STATE_ORDER:
		fbAdsWrite();
		IF NOT fbAdsWrite.BUSY THEN
			IF fbAdsWrite.Err THEN
				Error := TRUE;
				ErrorID := fbAdsWrite.ErrId;
				fbAdsWrite(WRITE := FALSE);
				iState := STATE_INITIALIZATION;
			ELSE
				IF  (Slave.NcToPlc.CoupleState < 2) THEN
					(* axis successfully decoupled *)
					Done := TRUE;
					iState := STATE_INITIALIZATION;
				ELSE (* wait for Nc2Plc feedback *)
					(* Done := TRUE; *)					 (* removed 2012-12-22 KSt *)
					(* iState := STATE_INITIALIZATION; *)	 (* removed 2012-12-22 KSt *)
					iState := STATE_RUNNING;			 (* added 2012-12-22 KSt *)
				END_IF
				fbAdsWrite(WRITE := FALSE);
			END_IF;
		END_IF;

	STATE_RUNNING:  (* waiting for Nc2Plc feedback - added 2012-12-22 KSt *)
		TimerStateFeedback(IN:=TRUE, PT:=t#50ms);
		IF  (Slave.NcToPlc.CoupleState < 2) THEN
			(* axis successfully decoupled *)
			Done := TRUE;
			iState := STATE_INITIALIZATION;
		ELSIF TimerStateFeedback.Q THEN
			(* 	nCoupleState does not respond 'not coupled' 	*)
			Error := TRUE;
			ErrorID := MC_ERROR_STATE_FEEDBACK_TIMEOUT;
			iState := STATE_INITIALIZATION;
		END_IF;

	ELSE  (* CASE : Unknown program state *)
		Error := TRUE;
		ErrorID := 16#FFFFFFFF;
		iState:= STATE_INITIALIZATION;
END_CASE

ADSbusy := fbAdsWrite.BUSY;

IF iState=STATE_INITIALIZATION THEN
	(* reset Busy immediately  when sequence ends *)
	IF Busy THEN
		LastExecutionResult.Done := Done;
		LastExecutionResult.Error := Error;
		LastExecutionResult.ErrorID := ErrorID;
	END_IF
	Busy := FALSE;
END_IF

END_FUNCTION_BLOCK

// POUs/Motion/Manual Motion/MC_Jog
FUNCTION_BLOCK MC_Jog
(*	This function block commands a jogged movement to an axis.*)
VAR_IN_OUT
	Axis				:	AXIS_REF; (*Reference to an axis*)
END_VAR
VAR_INPUT
	JogForward 		: 	BOOL;
	JogBackwards 	: 	BOOL;
	Mode			: 	E_JogMode;
	Position 			: 	LREAL;
	Velocity			:	LREAL;
	Acceleration		:	LREAL;
	Deceleration		:	LREAL;
	Jerk				:	LREAL;
(*	BufferMode		:	MC_BufferMode;*)(* E *)
END_VAR
VAR_OUTPUT
	Done			:	BOOL;
	Busy 			:	BOOL;
	Active 			:	BOOL;
	CommandAborted	:	BOOL;
	Error			:	BOOL;
{attribute 'displaymode':='hex'}
	ErrorID			:	UDINT;
END_VAR
VAR
	state: INT;
	LastExecutionResult: _ST_FunctionBlockResults;
	StateDWord: BOOL;
END_VAR
{library private}
VAR
	ExecuteMoveVelocity: BOOL;
	MoveVelocity: MC_MoveVelocity;
	MoveVelocityOut : ST_McOutputs;
	Direction: MC_Direction;

	ExecuteHalt: BOOL;
	Halt: MC_Halt;
	HaltOut : ST_McOutputs;

	ExecuteMoveAbsolute: BOOL;
	MoveAbsolute: MC_MoveAbsolute;
	MoveAbsoluteOut : ST_McOutputs;

	ExecuteMoveRelative: BOOL;
	MoveRelative : MC_MoveRelative;
	MoveRelativeOut : ST_McOutputs;

	JogMove: _FB_MoveUniversalGeneric;
	LastJogMoveResult: _ST_FunctionBlockResults;
	ExecuteJogMove: BOOL;
	StartType: _E_TCNC_StartPosType;
	JogMoveOut : ST_McOutputs;

	JogEnd: BOOL;
	TargetPosition: LREAL;
	modulo: LREAL;
	moduloremainder: LREAL;
END_VAR

ActCheckJogEnd();

CASE state OF
	0 : (* Initialization *)
		Busy := FALSE;
		Active := FALSE;
		ExecuteMoveVelocity := FALSE;
		ExecuteMoveRelative := FALSE;
		ExecuteMoveAbsolute := FALSE;
		ExecuteJogMove := FALSE;
		ExecuteHalt := FALSE;

		IF NOT JogForward AND NOT JogBackwards THEN (* 2009-03-12 *)
			Done := FALSE;
			CommandAborted := FALSE;
			Error := FALSE;
			ErrorID := 0;
		ELSIF (JogForward OR JogBackwards) AND F_AxisInProtectedMode(Axis.NcToPlc.StateDWord) THEN(* 2009-11-18 KSt *)
			(* MC_Jog cannot be used in protected mode (e. g. slave axis) *)
			Error := TRUE;
			ErrorID := MC_ERROR_AXIS_IN_PROTECTED_MODE;
		ELSIF JogForward AND NOT JogBackwards THEN
			Done := FALSE;
			Busy := TRUE;
			CommandAborted := FALSE;
			Error := FALSE;
			ErrorID := 0;
			Direction := MC_Positive_Direction;
			CASE Mode OF
				MC_JOGMODE_STANDARD_SLOW :
					StartType := TCNC_START_ENDLESSPLUS_SLOWMANUAL;
					ExecuteJogMove := TRUE;
					state := 3;
				MC_JOGMODE_STANDARD_FAST :
					StartType := TCNC_START_ENDLESSPLUS_FASTMANUAL;
					ExecuteJogMove := TRUE;
					state := 3;
				MC_JOGMODE_CONTINOUS :
					ExecuteMoveVelocity := TRUE;
					state := 1;
				MC_JOGMODE_INCHING :
					TargetPosition := Position;
					ExecuteMoveRelative := TRUE;
					state := 4;
				MC_JOGMODE_INCHING_MODULO :
					// 2022-11-08 KSt - calculation changed
					// TargetPosition := Axis.NcToPlc.SetPos - Axis.NcToPlc.ModuloSetPos + Position;
					modulo := SEL(Position=0, Position, 360); // 360 default
					moduloremainder := modabs(Axis.NcToPlc.SetPos, modulo);
					IF ABS(moduloremainder) < 1E-6 OR ABS(moduloremainder-modulo) < 1E-6 THEN
						// very close to a modulo limit 
						TargetPosition := Axis.NcToPlc.SetPos + modulo; // relative to current position value
					ELSE
						// position away from a modulo limit - adjust to modulo
						TargetPosition := modturns(Axis.NcToPlc.SetPos, modulo) * modulo + modulo;
					END_IF
					ExecuteMoveAbsolute := TRUE;
					state := 2;
			ELSE
				Busy := FALSE;
			END_CASE
		ELSIF JogBackwards AND NOT JogForward THEN
			Done := FALSE;
			Busy := TRUE;
			CommandAborted := FALSE;
			Error := FALSE;
			ErrorID := 0;
			Direction := MC_Negative_Direction;
			CASE Mode OF
				MC_JOGMODE_STANDARD_SLOW :
					StartType := TCNC_START_ENDLESSMINUS_SLOWMANUAL;
					ExecuteJogMove := TRUE;
					state := 3;
				MC_JOGMODE_STANDARD_FAST :
					StartType := TCNC_START_ENDLESSMINUS_FASTMANUAL;
					ExecuteJogMove := TRUE;
					state := 3;
				MC_JOGMODE_CONTINOUS :
					ExecuteMoveVelocity := TRUE;
					state := 1;
				MC_JOGMODE_INCHING :
					TargetPosition := - Position;
					ExecuteMoveRelative := TRUE;
					state := 4;
				MC_JOGMODE_INCHING_MODULO :
					// 2022-11-08 KSt - calculation changed
					(*
					modulo := Axis.NcToPlc.ModuloSetPos;
					IF modulo = 0 THEN
						TargetPosition := Axis.NcToPlc.SetPos - Position;
					ELSE
						TargetPosition := Axis.NcToPlc.SetPos - Axis.NcToPlc.ModuloSetPos;
					END_IF
					*)
					modulo := SEL(Position=0, Position, 360); // 360 default
					moduloremainder := modabs(Axis.NcToPlc.SetPos, modulo);
					IF ABS(moduloremainder) < 1E-6 OR ABS(moduloremainder-modulo) < 1E-6 THEN
						// very close to a modulo limit 
						TargetPosition := Axis.NcToPlc.SetPos - modulo; // relative to current position value
					ELSE
						// position away from a modulo limit - adjust to modulo
						TargetPosition := modturns(Axis.NcToPlc.SetPos, modulo) * modulo; // don't add or substract anything
					END_IF
					ExecuteMoveAbsolute := TRUE;
					state := 2;
			ELSE
				Busy := FALSE;
			END_CASE
		END_IF

	1 : (* continous jogging with MoveVelocity *)
		IF JogEnd THEN
			ExecuteMoveVelocity := FALSE;
			ExecuteHalt := TRUE;
		END_IF
		IF NOT MoveVelocity.Busy AND NOT Halt.Busy AND NOT F_AxisHasJob(Axis.NcToPlc.StateDWord) THEN
			Error := MoveVelocity.Error OR Halt.Error OR F_AxisInErrorState(Axis.NcToPlc.StateDWord);
			ErrorID := SEL( F_AxisInErrorState(Axis.NcToPlc.StateDWord), SEL(MoveVelocity.Error, Halt.ErrorID, MoveVelocity.ErrorID ), Axis.NcToPlc.ErrorCode);
			CommandAborted := NOT Error AND MoveVelocity.CommandAborted AND NOT ExecuteHalt; (* logic fixed 14.3.07 KSt *)
			Done := NOT Error AND NOT CommandAborted;
			ExecuteMoveVelocity := FALSE;
			ExecuteHalt := FALSE;
			IF JogEnd OR Done THEN
				state := 0;
			ELSE
				state := 9;
			END_IF
		END_IF

	2 : (* inching with MoveAbsolute *)
		IF 	Done OR
			(NOT MoveAbsolute.Busy AND NOT F_AxisHasJob(Axis.NcToPlc.StateDWord)) THEN
			Error := MoveAbsolute.Error;
			ErrorID := MoveAbsolute.ErrorID;
			CommandAborted := MoveAbsolute.CommandAborted;
			Done := NOT Error AND NOT CommandAborted;
			ExecuteMoveAbsolute := FALSE;
			IF JogEnd THEN
				state := 0;
			ELSE
				state := 9;
			END_IF
		END_IF

	3 : (* continous jogging with system parameters *)
		IF JogEnd THEN
			ExecuteJogMove := FALSE;
			ExecuteHalt := TRUE;
		END_IF
		IF NOT JogMove.Busy AND NOT Halt.Busy AND NOT F_AxisHasJob(Axis.NcToPlc.StateDWord) THEN
			Error := JogMove.Error OR Halt.Error OR F_AxisInErrorState(Axis.NcToPlc.StateDWord);
			ErrorID := SEL( F_AxisInErrorState(Axis.NcToPlc.StateDWord), SEL(JogMove.Error, Halt.ErrorID, JogMove.ErrorID ), Axis.NcToPlc.ErrorCode);
			CommandAborted := NOT Error AND JogMove.CommandAborted AND NOT ExecuteHalt; (* logic fixed 14.3.07 KSt *)
			Done := NOT Error AND NOT CommandAborted;
			ExecuteJogMove := FALSE;
			ExecuteHalt := FALSE;
			IF JogEnd OR Done THEN
				state := 0;
			ELSE
				state := 9;
			END_IF
		END_IF

	4 : (* inching with MoveRelative *)
		IF 	Done OR
			(NOT MoveRelative.Busy AND NOT F_AxisHasJob(Axis.NcToPlc.StateDWord)) THEN
			Error := MoveRelative.Error;
			ErrorID := MoveRelative.ErrorID;
			CommandAborted := MoveRelative.CommandAborted;
			Done := NOT Error AND NOT CommandAborted;
			ExecuteMoveRelative := FALSE;
			IF JogEnd THEN
				state := 0;
			ELSE
				state := 9;
			END_IF
		END_IF

	9 :	(* wait for falling edge on execute *)
		IF JogEnd THEN
			state := 0;
		END_IF
END_CASE

ActJogMove();

IF state = 0 OR state = 9 THEN
	IF Busy THEN
		LastExecutionResult.Done := Done;
		LastExecutionResult.CommandAborted := CommandAborted;
		LastExecutionResult.Error := Error;
		LastExecutionResult.ErrorID := ErrorID;
	END_IF
	Busy := FALSE;
	Active := FALSE;
ELSIF F_AxisInProtectedMode(Axis.NcToPlc.StateDWord) THEN (* 2009-11-18 KSt *)
	(* if axis is coupled on the fly - force state machine back to state zero and signal an error *)
	state := 0;
	Error := TRUE;
	ErrorID := MC_ERROR_AXIS_IN_PROTECTED_MODE;
END_IF

ACTION ActCheckJogEnd:
JogEnd := 	(NOT JogForward AND NOT JogBackwards) OR
			(NOT JogForward AND Direction=MC_Positive_Direction) OR
			(NOT JogBackwards AND Direction=MC_Negative_Direction);
END_ACTION

ACTION ActJogMove:
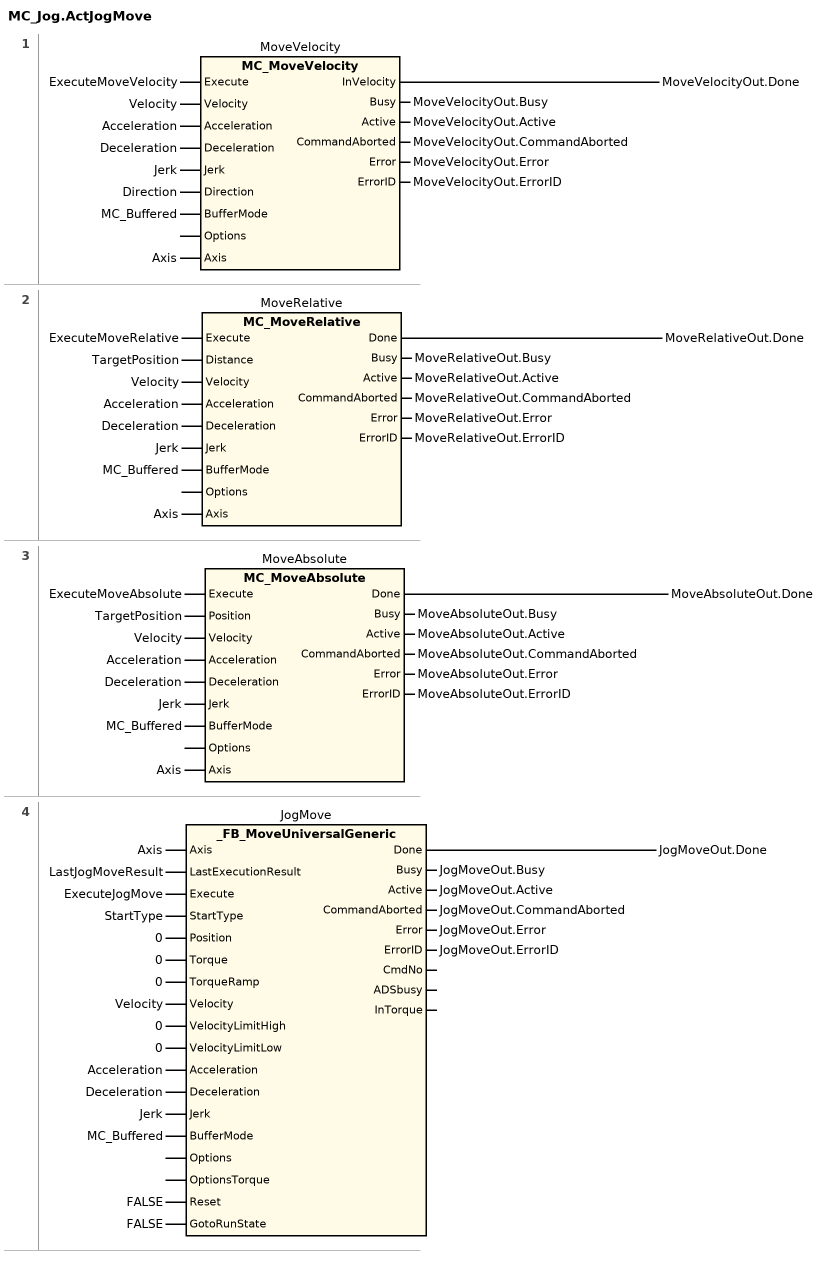
// NETWORK 1
MoveVelocity(
    Execute := ExecuteMoveVelocity,
    Velocity := Velocity,
    Acceleration := Acceleration,
    Deceleration := Deceleration,
    Jerk := Jerk,
    Direction := Direction,
    BufferMode := MC_Buffered,
    Axis := Axis,
    Busy => MoveVelocityOut.Busy,
    Active => MoveVelocityOut.Active,
    CommandAborted => MoveVelocityOut.CommandAborted,
    Error => MoveVelocityOut.Error,
    ErrorID => MoveVelocityOut.ErrorID); // MC_MoveVelocity
MoveVelocityOut.Done := MoveVelocity.InVelocity;

// NETWORK 2
MoveRelative(
    Execute := ExecuteMoveRelative,
    Distance := TargetPosition,
    Velocity := Velocity,
    Acceleration := Acceleration,
    Deceleration := Deceleration,
    Jerk := Jerk,
    BufferMode := MC_Buffered,
    Axis := Axis,
    Busy => MoveRelativeOut.Busy,
    Active => MoveRelativeOut.Active,
    CommandAborted => MoveRelativeOut.CommandAborted,
    Error => MoveRelativeOut.Error,
    ErrorID => MoveRelativeOut.ErrorID); // MC_MoveRelative
MoveRelativeOut.Done := MoveRelative.Done;

// NETWORK 3
MoveAbsolute(
    Execute := ExecuteMoveAbsolute,
    Position := TargetPosition,
    Velocity := Velocity,
    Acceleration := Acceleration,
    Deceleration := Deceleration,
    Jerk := Jerk,
    BufferMode := MC_Buffered,
    Axis := Axis,
    Busy => MoveAbsoluteOut.Busy,
    Active => MoveAbsoluteOut.Active,
    CommandAborted => MoveAbsoluteOut.CommandAborted,
    Error => MoveAbsoluteOut.Error,
    ErrorID => MoveAbsoluteOut.ErrorID); // MC_MoveAbsolute
MoveAbsoluteOut.Done := MoveAbsolute.Done;

// NETWORK 4
JogMove(
    Axis := Axis,
    LastExecutionResult := LastJogMoveResult,
    Execute := ExecuteJogMove,
    StartType := StartType,
    Position := 0,
    Torque := 0,
    TorqueRamp := 0,
    Velocity := Velocity,
    VelocityLimitHigh := 0,
    VelocityLimitLow := 0,
    Acceleration := Acceleration,
    Deceleration := Deceleration,
    Jerk := Jerk,
    BufferMode := MC_Buffered,
    Reset := FALSE,
    GotoRunState := FALSE,
    Busy => JogMoveOut.Busy,
    Active => JogMoveOut.Active,
    CommandAborted => JogMoveOut.CommandAborted,
    Error => JogMoveOut.Error,
    ErrorID => JogMoveOut.ErrorID); // _FB_MoveUniversalGeneric
JogMoveOut.Done := JogMove.Done;

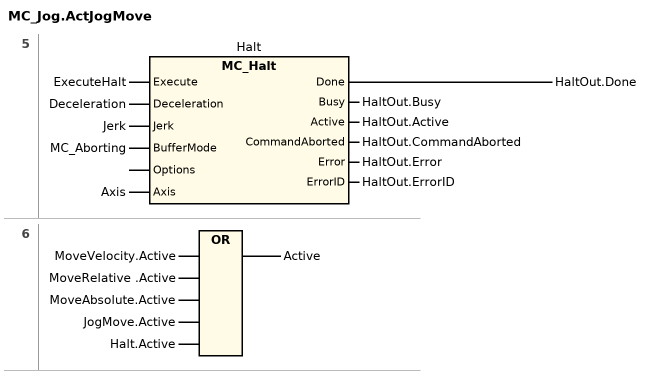
// NETWORK 5
Halt(
    Execute := ExecuteHalt,
    Deceleration := Deceleration,
    Jerk := Jerk,
    BufferMode := MC_Aborting,
    Axis := Axis,
    Busy => HaltOut.Busy,
    Active => HaltOut.Active,
    CommandAborted => HaltOut.CommandAborted,
    Error => HaltOut.Error,
    ErrorID => HaltOut.ErrorID); // MC_Halt
HaltOut.Done := Halt.Done;

// NETWORK 6
Active := MoveVelocity.Active OR (MoveRelative .Active) OR MoveAbsolute.Active OR JogMove.Active OR Halt.Active;
END_ACTION

END_FUNCTION_BLOCK

// POUs/Motion/Superposition/MC_AbortSuperposition
FUNCTION_BLOCK MC_AbortSuperposition
VAR_INPUT
	Execute		:	BOOL;	(* Starts touch probe recording *)
END_VAR
VAR_OUTPUT
	Done		:	BOOL;	(* move completed *)
	Busy		: 	BOOL;	(* function block is currently Busy *)
	Error		:	BOOL;	(* Signals that error has occured within Function Block *)
{attribute 'displaymode':='hex'}
	ErrorID		:	UDINT;	(* Error identification *)
END_VAR
VAR_IN_OUT
	Axis			:	AXIS_REF; (*Reference to an axis*)
END_VAR
VAR
	LastExecutionResult: 	_ST_FunctionBlockResults;
	ADSbusy	: 	BOOL;
	fbOnTrigger	: 	R_TRIG;
	fbADSwrite	: 	ADSWRITE;
	iState		:	_E_TcMC_STATES := STATE_INITIALIZATION;
END_VAR

fbOnTrigger(CLK:= Execute);

CASE iState OF
STATE_INITIALIZATION: (* initial iState *)
	Busy := FALSE;
	IF NOT Execute THEN
		Done := FALSE;
		Error := FALSE;
		ErrorID := 0;
	END_IF
	IF fbOnTrigger.Q THEN
		Busy := TRUE;
		(* initialization *)
		Done := FALSE;
		Error := FALSE;
		ErrorID := 0;
		LastExecutionResult.Done := FALSE;
		LastExecutionResult.CommandAborted := FALSE;
		LastExecutionResult.Error := FALSE;
		LastExecutionResult.ErrorID := 0;
		fbADSwrite(WRITE:=FALSE);
		fbADSwrite(	NETID:= TcMcGlobal.NCNETID_TCMC,
					(* PORT:=TcMcGlobal.NCPORT_TCMC , *)		(* 20140930 KSt *)
					PORT:=TcMcGlobal.NCPORT_TCMC_SUPERPOSITION,	(* 20140930 KSt *)
					IDXGRP:= TcMcGlobal.Axis.Functions.IDXGRP + Axis.NcToPlc.AxisId,
					IDXOFFS:= TcMcGlobal.Axis.Functions.IDXOFFS.STOPSCOM,	(* abort superposition *)
					LEN:=0,
					SRCADDR:=0,
					WRITE:=TRUE ,
					TMOUT:= TcMcGlobal.tADSTimeOut);
		iState := STATE_ORDER;
	END_IF

STATE_ORDER:  (* wait until command is accepted *)
	fbADSwrite(WRITE:= TRUE);
	IF NOT fbADSwrite.BUSY THEN
		Error := fbADSwrite.ERR;
		ErrorID := fbADSwrite.ERRID;
		IF NOT Error THEN
			IF NOT F_AxisIsCompensating(Axis.NcToPlc.StateDWord) THEN
				Done := TRUE;
				Busy := FALSE;
				iState := STATE_INITIALIZATION;
			ELSE
				iState := STATE_RUNNING;
			END_IF
		ELSE
			Busy := FALSE;
			iState := STATE_INITIALIZATION;
		END_IF
		LastExecutionResult.Done := Done;
		LastExecutionResult.Error := Error;
		LastExecutionResult.ErrorID := ErrorID;
	END_IF

STATE_RUNNING:
	IF NOT F_AxisIsCompensating(Axis.NcToPlc.StateDWord) THEN
		Done := TRUE;
		Busy := FALSE;
		LastExecutionResult.Done := Done;
		LastExecutionResult.Error := Error;
		LastExecutionResult.ErrorID := ErrorID;
		iState := STATE_INITIALIZATION;
	END_IF
END_CASE

ADSbusy := fbAdsWrite.BUSY;

END_FUNCTION_BLOCK

// POUs/Motion/Gearing/MC_GearInMultiMaster
FUNCTION_BLOCK MC_GearInMultiMaster
(*	MC_GearInDyn couples a slave axis to a master axis
 *	using a floating point gear ratio. The gear ratio can be 
 *	dynamically modified every PLC cycle as long as the 
 *	Execute input is TRUE.
 *	The acceleration input specifies the maximum slave
 *	acceleration in case of high gear ratio changes.
 *)
VAR_INPUT
 {attribute 'init_on_onlchange'}
	Master1: REFERENCE TO AXIS_REF; (*Reference to an axis*)
 {attribute 'init_on_onlchange'}
	Master2: REFERENCE TO AXIS_REF; (*Reference to an axis*)
 {attribute 'init_on_onlchange'}
	Master3: REFERENCE TO AXIS_REF; (*Reference to an axis*)
 {attribute 'init_on_onlchange'}
	Master4: REFERENCE TO AXIS_REF; (*Reference to an axis*)
END_VAR
VAR_IN_OUT
	Slave: AXIS_REF; (*Reference to an axis*)
END_VAR
VAR_INPUT
	Enable			:	BOOL;
	GearRatio1		:	LREAL := 1.0;
	GearRatio2		:	LREAL := 1.0;
	GearRatio3		:	LREAL := 1.0;
	GearRatio4		:	LREAL := 1.0;
{attribute 'conditionalshow'}
	Velocity		:	LREAL;	// Velocity added - 20220518 KSt
	Acceleration	:	LREAL;
	Deceleration	:	LREAL;	(* just used in version 2 mode (AdvancedSlaveDynamics) *)
	Jerk			:	LREAL;	(* just used in version 2 mode (AdvancedSlaveDynamics) *)
	BufferMode		:	MC_BufferMode;	(* E *)
	Options			: 	ST_GearInMultiMasterOptions;	(* V *)	(* optional parameters *)
END_VAR
VAR_OUTPUT
	InGear				:	BOOL;
	Busy				: 	BOOL;
	Active				: 	BOOL;
	CommandAborted		:	BOOL;
	Error				:	BOOL;
{attribute 'displaymode':='hex'}
	ErrorID				:	UDINT;
END_VAR
VAR
	InGear2				:	BOOL;
	ADSbusy				: 	BOOL;
	iState				:	_E_TcMC_STATES := STATE_INITIALIZATION;
	fbAdsWrite			:	ADSWRITE;
	sCouple				:	_ST_TcNC_CoupleSlaveMultiMaster;
	sCoupleV2			:	_ST_TcNC_CoupleSlaveMultiMaster2;
	LastExecutionResult	: 	_ST_FunctionBlockResults;
	IsCoupled			: 	BOOL;
	LastNcCycleCounter	:	BYTE;
{attribute 'conditionalshow'}
	InGear2Cnt			: UDINT;
{attribute 'conditionalshow'}
	i					: UDINT;
END_VAR
VAR
{attribute 'conditionalshow'}
	TimerStateFeedback		: 	TON;
{attribute 'conditionalshow'}
	iAdvancedSlaveDynamics	:	BOOL;
{attribute 'conditionalshow'}
	iVelocity				: 	LREAL;
{attribute 'conditionalshow'}
	iAcceleration			: 	LREAL;
{attribute 'conditionalshow'}
	iDeceleration			:	LREAL;	(* just used in version 2 mode *)
{attribute 'conditionalshow'}
	iJerk					:	LREAL;	(* just used in version 2 mode *)
{attribute 'conditionalshow'}
	iGearRatio1				:	LREAL := 1.0;
{attribute 'conditionalshow'}
	iGearRatio2				:	LREAL := 1.0;
{attribute 'conditionalshow'}
	iGearRatio3				:	LREAL := 1.0;
{attribute 'conditionalshow'}
	iGearRatio4				:	LREAL := 1.0;
{attribute 'conditionalshow'}
	WasInGear				:	 BOOL;
{attribute 'conditionalshow'}
	GearRatioChanged		:	 BOOL;
{attribute 'conditionalshow'}
	ParameterChanged		:	 BOOL;
{attribute 'conditionalshow'}
	GearRatioChangePending	:	 BOOL;
END_VAR

IF NOT _F_TcMC_IsValidAxisRef(Slave) THEN // AXIS REFERENCE CHECK - 2020-09-17 KSt
	Error := TRUE;
	ErrorID := MC_ERROR_INVALIDREFERENCE;
	RETURN;
END_IF

IF Enable AND NOT Busy THEN
	(* AdvancedSlaveDynamics can only be changed when triggered *)
	iAdvancedSlaveDynamics := Options.AdvancedSlaveDynamics;
END_IF

IF iAdvancedSlaveDynamics THEN
	ActGearInMultiMasterV2();	(* new version V2 - 2011-09-07 KSt *)
ELSE
	ActGearInMultiMasterV1();	(* classic version V1 *)
END_IF

ACTION ActGearInMultiMasterV1:
(*
 *	CLASSIC   MC_GearInMultimaster 
 *)
CASE iState OF
	STATE_INITIALIZATION:	(* *)
		Busy := FALSE;
		Active := FALSE;
		IF Enable THEN
			Busy := TRUE;
			Active := TRUE;
			fbAdsWrite(WRITE:=FALSE);
			(* initialize output values *)
			iAcceleration := Acceleration;
			ErrorID := 0;
			Error := FALSE;
			LastExecutionResult.Done := FALSE;
			LastExecutionResult.CommandAborted := FALSE;
			LastExecutionResult.Error := FALSE;
			LastExecutionResult.ErrorID := 0;
			TimerStateFeedback(IN:=FALSE);
			WasInGear := FALSE;

			IF BufferMode <> 0 THEN
				Error := TRUE;
				ErrorID := MC_ERROR_BUFFERMODE_NOT_SUPPORTED;
			ELSIF NOT __ISVALIDREF(Master1)
			  AND NOT __ISVALIDREF(Master2)
			  AND NOT __ISVALIDREF(Master3)
			  AND NOT __ISVALIDREF(Master4) THEN
				Error := TRUE;
				ErrorID := MC_ERROR_PARAMETER_NOT_CORRECT;
			ELSE
				InGear := F_AxisIsCoupled(Slave.NcToPlc.CoupleState) ;
				istate := SEL( InGear, STATE_ORDER, STATE_RUNNING);
			END_IF

		ELSE
			// FAP 2018-07-12 Initialize references only while ENABLE = FALSE
			Master1 REF= 0;
			Master2 REF= 0;
			Master3 REF= 0;
			Master4 REF= 0;	
			Error := FALSE;	(* reset when Enable is FALSE *)
			ErrorID := 0;
			CommandAborted := FALSE;
			InGear := FALSE;
		END_IF

	STATE_ORDER :
			(* couple with dynamic gear ratio *)
			sCouple.nSlaveType := INT_TO_UDINT(TCNC_SLAVETYPE_LINEAR_MULTIMASTER);
			sCouple.nMasterSubIdx	:= 0;
			sCouple.nSlaveSubIdx		:= 0;
(*			sCouple.fCoupleParam1	:= iAcceleration;*)

			//	FAP 2017-09-07 Master1-4 are now optional references to AXIS_REF / validation check in needed to avoid access to not referenced adresses
			sCouple.nMasterAxisId := SEL(__ISVALIDREF(Master1), 0, Master1.NcToPlc.AxisId);;
			sCouple.nMasterID2 := SEL(__ISVALIDREF(Master2), 0, Master2.NcToPlc.AxisId);;
			sCouple.nMasterID3 := SEL(__ISVALIDREF(Master3), 0, Master3.NcToPlc.AxisId);;
			sCouple.nMasterID4 := SEL(__ISVALIDREF(Master4), 0, Master4.NcToPlc.AxisId);;
			//sCouple.nMasterAxisId := Master1.NcToPlc.AxisId
			//sCouple.nMasterID2 := Master2.NcToPlc.AxisId;
			//sCouple.nMasterID3 := Master3.NcToPlc.AxisId;
			//sCouple.nMasterID4 := Master4.NcToPlc.AxisId;

			sCouple.fSlaveAcceleration := iAcceleration;
(* 			sCouple.nCheckAndOpMode := ? *)

			(* cyclic data *)
			Slave.PlcToNc.GearRatio1 := GearRatio1;
			Slave.PlcToNc.GearRatio2 := GearRatio2;
			Slave.PlcToNc.GearRatio3 := GearRatio3;
			Slave.PlcToNc.GearRatio4 := GearRatio4;

			fbAdsWrite(	NETID:= TcMcGlobal.NCNETID_TCMC,
					PORT:= TcMcGlobal.NCPORT_TCMC_COUPLING,
					IDXGRP:=TcMcGlobal.Axis.Functions.IDXGRP+Slave.NcToPlc.AxisId,
					IDXOFFS:= TcMcGlobal.Axis.Functions.IDXOFFS.CPL,
					LEN:= SIZEOF(sCouple),
					SRCADDR:= ADR(sCouple),
					WRITE:= TRUE,
					TMOUT:= TcMcGlobal.tADSTimeOut);
			IF NOT fbAdsWrite.Busy THEN
				Error := fbAdsWrite.ERR;
				ErrorID := fbAdsWrite.ERRID;
				fbAdsWrite(WRITE:=FALSE);
				IF Error THEN
					iState := STATE_INITIALIZATION;
				ELSE
					InGear := F_AxisIsCoupled(Slave.NcToPlc.CoupleState);
					iState := STATE_RUNNING;
				END_IF
			END_IF

	STATE_RUNNING:  (* cyclic change of the gear ratio until decoupled or until Execute=FALSE *)
		TimerStateFeedback(IN:=TRUE, PT:=t#50ms); (* 5.7.2006 KSt *)
		Slave.PlcToNc.GearRatio1 := GearRatio1;
		Slave.PlcToNc.GearRatio2 := GearRatio2;
		Slave.PlcToNc.GearRatio3 := GearRatio3;
		Slave.PlcToNc.GearRatio4 := GearRatio4;
		InGear := F_AxisIsCoupled(Slave.NcToPlc.CoupleState) ;
		IF InGear THEN
			WasInGear := TRUE; (* feedback seen, 5.7.2006 KSt *)
		END_IF
		IF (NOT Enable OR NOT InGear) AND (WasInGear OR TimerStateFeedback.Q) THEN (* 5.7.2006 KSt *)
(*  keep latest gear ratio - 2008-02-19 KSt *)
			(* stop when still in gear but not enabled *)
(*			Slave.PlcToNc.GearRatio1 := 0;
			Slave.PlcToNc.GearRatio2 := 0;
			Slave.PlcToNc.GearRatio3 := 0;
			Slave.PlcToNc.GearRatio4 := 0;
*)
			CommandAborted := NOT InGear;
			iState := STATE_INITIALIZATION;
		END_IF;

	ELSE  (* CASE : Unknown program state *)
		Error := TRUE;
		ErrorID := 16#FFFFFFFF;
		iState:= STATE_INITIALIZATION;
END_CASE

ADSbusy := fbAdsWrite.BUSY;
IF iState=STATE_INITIALIZATION THEN
	(* reset Busy immediately  when sequence ends *)
	IF Busy THEN
		LastExecutionResult.Done := InGear;
		LastExecutionResult.CommandAborted := CommandAborted;
		LastExecutionResult.Error := Error;
		LastExecutionResult.ErrorID := ErrorID;
	END_IF
	Busy := FALSE;
	Active := FALSE;
END_IF
END_ACTION

ACTION ActGearInMultiMasterV2:
(*
 *	EXTENDED   MC_GearInMultimaster Version 2
 *	2011-09-07 KSt 
 *)
 FOR i := 1 TO 2 DO (* 29.09.2015 FAP *)
	CASE iState OF
		STATE_INITIALIZATION:	(* *)
			Busy := FALSE;
			Active := FALSE;
			IF Enable THEN
				Busy := TRUE;
				Active := TRUE;
				fbAdsWrite(WRITE:=FALSE);
				(* initialize output values *)
				iVelocity := Velocity;	// Velocity added - 20220518 KSt
				iAcceleration := Acceleration;
				iDeceleration := Deceleration;
				iJerk := Jerk;
				iGearRatio1	:= GearRatio1;
				iGearRatio2 := GearRatio2;
				iGearRatio3 := GearRatio3;
				iGearRatio4 := GearRatio4;
				
				GearRatioChangePending := FALSE;
				ErrorID := 0;
				Error := FALSE;
				LastExecutionResult.Done := FALSE;
				LastExecutionResult.CommandAborted := FALSE;
				LastExecutionResult.Error := FALSE;
				LastExecutionResult.ErrorID := 0;
				TimerStateFeedback(IN:=FALSE);
				WasInGear := FALSE;
	
				IF BufferMode <> 0 THEN
					Error := TRUE;
					ErrorID := MC_ERROR_BUFFERMODE_NOT_SUPPORTED;
					EXIT;
				ELSE
					IsCoupled := F_AxisIsCoupled(Slave.NcToPlc.CoupleState) ;
					istate := SEL( IsCoupled, STATE_ORDER, STATE_RUNNING);
					IF iState = STATE_ORDER THEN (* 02.10.2015 FAP *)
						Slave.PlcToNc.GearRatio1 := GearRatio1;
						Slave.PlcToNc.GearRatio2 := GearRatio2;
						Slave.PlcToNc.GearRatio3 := GearRatio3;
						Slave.PlcToNc.GearRatio4 := GearRatio4;
						EXIT;
					END_IF
				END_IF
			ELSE
				// FAP 2018-07-12 Initialize references only while ENABLE = FALSE
				Master1 REF= 0;
				Master2 REF= 0;
				Master3 REF= 0;
				Master4 REF= 0;	
				Error := FALSE;	(* reset when Enable is FALSE *)
				ErrorID := 0;
				CommandAborted := FALSE;
				InGear := FALSE;
				InGear2 := FALSE;(* 29.09.2015 FAP *)
				EXIT;
			END_IF
	
		STATE_ORDER :
			IsCoupled := F_AxisIsCoupled(Slave.NcToPlc.CoupleState) ;
			InGear := Slave.NcToPlc.AxisState=INT_TO_DWORD(TCNC_PHASE_SYNCHRONOUS);
			InGear2 := FALSE; (* 29.09.2015 FAP *)
			(* couple with dynamic gear ratio *)
			sCoupleV2.nSlaveType := INT_TO_UDINT(TCNC_SLAVETYPE_LINEAR_MULTIMASTER);
			sCoupleV2.nMasterSubIdx	:= 0;
			sCoupleV2.nSlaveSubIdx	:= 0;
			IF NOT IsCoupled THEN
				//	FAP 2017-09-07 Master2-4 are now optional references to AXIS_REF / validation check in needed to avoid access to not referenced adresses
				sCoupleV2.nMasterAxisId := SEL(__ISVALIDREF(Master1), 0, Master1.NcToPlc.AxisId);;
				sCoupleV2.nMasterID2 := SEL(__ISVALIDREF(Master2), 0, Master2.NcToPlc.AxisId);;
				sCoupleV2.nMasterID3 := SEL(__ISVALIDREF(Master3), 0, Master3.NcToPlc.AxisId);;
				sCoupleV2.nMasterID4 := SEL(__ISVALIDREF(Master4), 0, Master4.NcToPlc.AxisId);;
				//sCoupleV2.nMasterAxisId := Master1.NcToPlc.AxisId;
				//sCoupleV2.nMasterID2 := Master2.NcToPlc.AxisId;
				//sCoupleV2.nMasterID3 := Master3.NcToPlc.AxisId;
				//sCoupleV2.nMasterID4 := Master4.NcToPlc.AxisId;
			END_IF
			// sCoupleV2.fSlaveMaxVelo := 0;	(* use axis default *)
			sCoupleV2.fSlaveMaxVelo := iVelocity;	// Velocity added - 20220518 KSt
			sCoupleV2.fSlaveMaxAcc := iAcceleration;
			sCoupleV2.fSlaveMaxDec := iDeceleration;
			sCoupleV2.fSlaveMaxJerk := iJerk;
			// sCoupleV2.nCheckAndOpMode.0 := Options.VelocitySynchronizationOnly;	(* set bit 0 in bit array *) // unused and deleted since 2020-05-27 KSt 
			CASE Options.SyncMode OF // new SyncMode since 2020-05-27 KSt
				E_GearInMultiMasterSyncMode.VELOSYNC : sCoupleV2.nCheckAndOpMode := 0;
				E_GearInMultiMasterSyncMode.POSSYNC1 : sCoupleV2.nCheckAndOpMode := 1;
				E_GearInMultiMasterSyncMode.POSSYNC2 : sCoupleV2.nCheckAndOpMode := 2;
			ELSE
				sCoupleV2.nCheckAndOpMode := 0 + 0;
			END_CASE
	
			(* cyclic data *)
			IF NOT GearRatioChangePending THEN	
				Slave.PlcToNc.GearRatio1 := GearRatio1;
				Slave.PlcToNc.GearRatio2 := GearRatio2;
				Slave.PlcToNc.GearRatio3 := GearRatio3;
				Slave.PlcToNc.GearRatio4 := GearRatio4;
			END_IF
			
			fbAdsWrite(	NETID:= TcMcGlobal.NCNETID_TCMC,
					PORT:= TcMcGlobal.NCPORT_TCMC_COUPLING,
					IDXGRP:=TcMcGlobal.Axis.Functions.IDXGRP+Slave.NcToPlc.AxisId,
					IDXOFFS:= TcMcGlobal.Axis.Functions.IDXOFFS.CPL,
					LEN:= SIZEOF(sCoupleV2),
					SRCADDR:= ADR(sCoupleV2),
					WRITE:= TRUE,
					TMOUT:= TcMcGlobal.tADSTimeOut);
			IF NOT fbAdsWrite.Busy THEN
				Error := fbAdsWrite.ERR;
				ErrorID := fbAdsWrite.ERRID;
				fbAdsWrite(WRITE:=FALSE);
				IF Error THEN
					iState := STATE_INITIALIZATION;
				ELSE
					(* 29.09.2015 FAP *)
					IF _F_NcNoOfCycleCounterUpdated(LastNcCycleCounter, Slave) >= 2 THEN
						InGear2Cnt := 2;
						InGear2 := Slave.NcToPlc.AxisState=INT_TO_DWORD(TCNC_PHASE_SYNCHRONOUS);
					ELSE
						InGear2Cnt := 1;
					END_IF
					iState := STATE_RUNNING;
				END_IF
			ELSE
				EXIT;
			END_IF

			(* 29.09.2015 FAP *)
			LastNcCycleCounter := DWORD_TO_BYTE(SHR(Slave.NcToPlc.OpModeDWord, 24));
	
		STATE_RUNNING:  (* cyclic change of the gear ratio until decoupled or until Execute=FALSE *)
			TimerStateFeedback(IN:=TRUE, PT:=t#50ms); (* 5.7.2006 KSt *)

			(* 29.09.2015 FAP *)
			IF (Slave.PlcToNc.GearRatio1 <> GearRatio1)
			  OR (Slave.PlcToNc.GearRatio2 <> GearRatio2)
			  OR (Slave.PlcToNc.GearRatio3 <> GearRatio3)
			  OR (Slave.PlcToNc.GearRatio4 <> GearRatio4) THEN
				InGear2 := FALSE;
				InGear2Cnt := 0;
				LastNcCycleCounter := DWORD_TO_BYTE(SHR(Slave.NcToPlc.OpModeDWord, 24));
			END_IF

			GearRatioChanged :=
				(Slave.PlcToNc.GearRatio1 <> GearRatio1) OR
			  	(Slave.PlcToNc.GearRatio2 <> GearRatio2) OR
			  	(Slave.PlcToNc.GearRatio3 <> GearRatio3) OR
			  	(Slave.PlcToNc.GearRatio4 <> GearRatio4);
				
			ParameterChanged :=
				(Velocity <> iVelocity) OR 	// Velocity added - 20220518 KSt
				(Acceleration <> iAcceleration) OR
				(Deceleration <> iDeceleration) OR
				(Jerk <> iJerk);
			
			IF GearRatioChanged AND NOT ParameterChanged AND NOT GearRatioChangePending THEN	
				Slave.PlcToNc.GearRatio1 := GearRatio1;
				Slave.PlcToNc.GearRatio2 := GearRatio2;
				Slave.PlcToNc.GearRatio3 := GearRatio3;
				Slave.PlcToNc.GearRatio4 := GearRatio4;
			ELSIF GearRatioChanged AND ParameterChanged AND NOT GearRatioChangePending THEN	
				iGearRatio1	:= GearRatio1;
				iGearRatio2 := GearRatio2;
				iGearRatio3 := GearRatio3;
				iGearRatio4 := GearRatio4;
				GearRatioChangePending := TRUE;
			ELSIF GearRatioChangePending THEN
				Slave.PlcToNc.GearRatio1 := iGearRatio1;
				Slave.PlcToNc.GearRatio2 := iGearRatio2;
				Slave.PlcToNc.GearRatio3 := iGearRatio3;
				Slave.PlcToNc.GearRatio4 := iGearRatio4;
				GearRatioChangePending := FALSE;
			END_IF
			
			IsCoupled := F_AxisIsCoupled(Slave.NcToPlc.CoupleState) ;
			InGear := Slave.NcToPlc.AxisState=INT_TO_DWORD(TCNC_PHASE_SYNCHRONOUS);

			(* 29.09.2015 FAP *)
			IF _F_NcCycleCounterUpdated(LastNcCycleCounter, Slave) AND InGear2Cnt < 2 THEN
				IF _F_NcNoOfCycleCounterUpdated(LastNcCycleCounter, Slave) >= 2 THEN
					InGear2Cnt := 2;
				ELSE
					InGear2Cnt := InGear2Cnt + 1;
				END_IF
				LastNcCycleCounter := DWORD_TO_BYTE(SHR(Slave.NcToPlc.OpModeDWord, 24));
			END_IF	
			
			IF InGear2Cnt >= 2 OR InGear2 THEN
				InGear2 := Slave.NcToPlc.AxisState=INT_TO_DWORD(TCNC_PHASE_SYNCHRONOUS);
			END_IF
			
			IF IsCoupled THEN
				WasInGear := TRUE; (* feedback seen, 5.7.2006 KSt *)
			END_IF
			IF (NOT Enable OR NOT IsCoupled) AND (WasInGear OR TimerStateFeedback.Q) THEN (* 5.7.2006 KSt *)
				CommandAborted := NOT IsCoupled;
				iState := STATE_INITIALIZATION;
			ELSE
				IF ParameterChanged THEN
					iVelocity := Velocity;	// Velocity added - 20220518 KSt
					iAcceleration := Acceleration;
					iDeceleration := Deceleration;
					iJerk := Jerk;
					istate := STATE_ORDER;
				ELSE
					EXIT;
				END_IF
			END_IF;
	
		ELSE  (* CASE : Unknown program state *)
			Error := TRUE;
			ErrorID := 16#FFFFFFFF;
			iState:= STATE_INITIALIZATION;
	END_CASE
END_FOR

ADSbusy := fbAdsWrite.BUSY;
IF iState=STATE_INITIALIZATION THEN
	(* reset Busy immediately  when sequence ends *)
	IF Busy THEN
		LastExecutionResult.Done := InGear;
		LastExecutionResult.CommandAborted := CommandAborted;
		LastExecutionResult.Error := Error;
		LastExecutionResult.ErrorID := ErrorID;
	END_IF
	Busy := FALSE;
	Active := FALSE;
END_IF
END_ACTION

END_FUNCTION_BLOCK

// POUs/Administrative/Extensions/MC_SetEncoderScalingFactor
FUNCTION_BLOCK MC_SetEncoderScalingFactor
(*
	This function can change the encoder scaling factor in stand-still or on the fly.
*)
VAR_IN_OUT
	Axis			:	AXIS_REF; (*Reference to an axis*)
END_VAR
VAR_INPUT
	Execute		:	BOOL;		(* Start setting position in axis *)
	ScalingFactor	:	LREAL;	(* Position unit [u] / EncoderIncrements *)
	Mode		: 	E_SetScalingFactorMode;	
	Options		:	ST_SetEncoderScalingOptions;	(* Beckhoff proprietary input *)
END_VAR
VAR_OUTPUT
	Done		:	BOOL;		(* Position has new value *)
	Busy		:	BOOL;		(* Shows that the Function Block is not finished *)
	Error		:	BOOL;		(* Signals that an error has occurred within the Function Block *)
{attribute 'displaymode':='hex'}
	ErrorID		:	UDINT;		(* Error identification *)
END_VAR
(*
	Note:
	RELATIVE means that the actual position of the axis is adjusted to the 
	new scaling factor value in a way that no position jump will occur.
	ABSOLUTE means that the scaling factor will be set without any 
	internal position offsets. In this case the actual position value of the 
	axis will jump instantaneously.
	When changing the scaling factor on the fly, RELATIVE mode is 
	supposed to be preferred.
*)
VAR
	ADSbusy	: 	BOOL;
	stSetEncoderSaclingFactor	:	_ST_TcNC_SetEncoderSaclingFactor;
	iState		:	_E_TcMC_STATES := STATE_INITIALIZATION;
	fbAdsWrite	:	ADSWRITE;
END_VAR
VAR
{attribute 'conditionalshow'}
	fbOnTrigger	:	R_TRIG;
END_VAR


fbOnTrigger(CLK:= Execute);

CASE iState OF
STATE_INITIALIZATION:
	Busy := FALSE;
	IF NOT Execute THEN
		Done := FALSE;
		Error := FALSE;			(* reset at falling edge of Execute *)
		ErrorID := 0;
	END_IF
	IF fbOnTrigger.Q THEN
		Busy := TRUE;
		(* initialize output values *)
		Done := FALSE;
		Error := FALSE;
		ErrorID := 0;
		fbAdsWrite(WRITE := FALSE);

		(* fill structure*)
		stSetEncoderSaclingFactor.fEncoderScalingFactor := ScalingFactor;
		stSetEncoderSaclingFactor.nEncoderScalingFactorType := Mode;
		stSetEncoderSaclingFactor.nCtrlWord.1 := SEL( Options.SelectEncoderIndex, FALSE, TRUE ); 	(* set bit 1 to explicitly select an encoder / control loop - KSt 2009-04-09 *)

		IF Options.SelectEncoderIndex THEN (* KSt 2009-04-09 *)
			(* select the user defined encoder/control loop explicitly *)
			fbAdsWrite.IDXOFFS:= TcMcGlobal.Axis.Functions.IDXOFFS.SETENCODERSCALING + Options.EncoderIndex * 16#00100000;
		ELSE
			(* select the encoder / control loop that is defined by the AXIS_REF interface
				0  	=  select active encoder / control loop		- used when standard AXIS_REF interface is used
				1..n 	=  explicit encoder / control loop selection 	- used when dedicated encoder AXIS_REF interface is used 		*)
			fbAdsWrite.IDXOFFS:= TcMcGlobal.Axis.Functions.IDXOFFS.SETENCODERSCALING + Axis.NcToPlc.ControlLoopIndex * 16#00100000;
		END_IF

		fbAdsWrite(	NETID:= TcMcGlobal.NCNETID_TCMC,
					PORT:= AMSPORT_R0_NCSAF,
					IDXGRP:=TcMcGlobal.Axis.Functions.IDXGRP+Axis.NcToPlc.AxisId,
(*					IDXOFFS:= TcMcGlobal.Axis.Functions.IDXOFFS.SETENCODERSCALING + Options.EncoderIndex * 16#100000,*) (* KSt 2009-04-09 - see selection above *)
					LEN:= SIZEOF(stSetEncoderSaclingFactor),
					SRCADDR:= ADR(stSetEncoderSaclingFactor),
					WRITE:= TRUE,
					TMOUT:= TcMcGlobal.tADSTimeOut);
		iState := STATE_ORDER;
	END_IF;

STATE_ORDER:
	fbAdsWrite();
	IF NOT fbAdsWrite.Busy THEN
		IF fbAdsWrite.Err THEN
			ErrorID := fbAdsWrite.ErrId;
			Error := TRUE;
		ELSE
			Done := TRUE;
		END_IF;
		fbAdsWrite(WRITE := FALSE);
		iState := STATE_INITIALIZATION;
	END_IF;

ELSE  (* CASE : Unknown program state *)
	Error := TRUE;
	ErrorID := 16#FFFFFFFF;
	iState:= STATE_INITIALIZATION;
END_CASE

ADSbusy := fbAdsWrite.BUSY;

IF iState=STATE_INITIALIZATION THEN
	(* reset Busy immediately  when sequence ends *)
	Busy := FALSE;
END_IF

END_FUNCTION_BLOCK

// POUs/Administrative/Extensions/MC_BacklashCompensation
(*==============================================================================*)
(* Name:	MC_BacklashCompensation												*)
(*		(based on _FB_PositionCorrectionTableLookup + MC_PositionCorrectionLimiter)	*)
(* Parameter: returns a compensation value depending on the position of the reference axis	*)
(*		Use the nc function PositionCompensation to compensate the backlash			*)
(*		1. the FB _FB_PositionCorrectionTableLookup calculates the backlash value		*)
(*		2. the FB MC_PositionCorrectionLimiter feed this correction value					*)
(*		into the NcToPlc.PositionCorrection variable									*)
(* Requirements: The 'Position Correction' feature must be enabled in the SystemManager 	*)
(*																				*)
(* Author:	 	HKP																	*)
(* Date:		19-July-2012															*)
(* last edit:	VER 0.0.4															*)
(*==============================================================================*)

FUNCTION_BLOCK MC_BacklashCompensation
VAR_IN_OUT
	Axis							: AXIS_REF; (*Reference to an axis*)
END_VAR
VAR_INPUT
	Enable						: BOOL;							(* switch to activate backlash compensation *)
	Backlash					: LREAL := DEFAULT_BACKLASHVALUE;	(* signed backlash value [mm] (when using default value the internal nc backlash value will be read by ADS and used in this FB) *)
	CompensationInPositiveDirection : BOOL;							(* compensation is just working in the selected working direction *)
																(* FALSE (default): backlash compensation must be done when driving in negative direction;  TRUE: backlash compensation must be done when driving in positive direction *)
	Ramp						: LREAL;							(* velocity limit for feeded backlash compensation (constant velocity and linear position sub profile for backlash compensation) [mm/s] (default:=0.0) *)
	DisableMode					: E_DisableMode;					(* disable mode defines whow to react in case of disabling: (0)=HOLD, (1)=RESET, ... *)
	Options						: ST_BacklashCompensationOptions;	(* optional parameters (NOT USED YET) *)
END_VAR
VAR_OUTPUT
	Enabled						: BOOL;
	Busy						: BOOL;
	Error						: BOOL;
{attribute 'displaymode':='hex'}
	ErrorID						: UDINT;
	CurrentBacklash				: LREAL;							(* current actual backlash value [mm] *)
	Limiting						: BOOL;							(* function block is currently limiting the Backlash Correction *)
END_VAR
VAR
	InternalEnable				: BOOL;							(* trick for internal FB handling *)
	state						: INT;
	GetThisTaskIndex				: GETCURTASKINDEX;
	CycleTime					: LREAL;								(* task cycle time [s] *)
	fbCalcBacklashCorrection		: _FB_PositionCorrectionTableLookup;	(* based on old 'FB_PositionCompensation' in TcNc.lib *)
	fbFeedBacklashCorrection		: MC_PositionCorrectionLimiter;			(* s.TcMC2.lib (original based on old 'FB_WritePositionCorrection' in TcNc.lib) *)
	CalcBacklashCorrOut			: ST_McOutputs;
	FeedBacklashCorrOut			: ST_McOutputs;
	ReadParameter				: MC_ReadParameter;
	iBacklash					: LREAL;
	InternalAcceleration			: LREAL;								(* input of FB 'MC_PositionCorrectionLimiter': 'Acceleration' [mm/s^2] *)
	InternalBacklashValue			: LREAL;								(* output of FB 'MC_PositionCorrectionLimiter': 'PositionCorrectionValue' [mm] *)
	InternalLimitingActive			: BOOL;								(* output of FB 'MC_PositionCorrectionLimiter': 'Limiting' [0/1] *)

	stPosCompParameter : ST_PositionCompensationTableParameter :=
								( MinPosition := -1.0E+12, MaxPosition :=1.0E+12, NoOfTableElements :=2, Direction := WorkDirectionNegative );

	stPosCompTable: ARRAY[0..1] OF ST_PositionCompensationTableElement := [
								( Position := -1.0E+12,	Compensation := 0.0 ),
								( Position := +1.0E+12,	Compensation := 0.0 ) ];
END_VAR


CASE state OF
	0 : (* init *)
		Busy := FALSE;
		Enabled := FALSE;
		IF Enable THEN
			IF NOT Axis.NcToPlc.OpModeDWord.20 THEN (* PositionCorrection active ? *)
				Error := TRUE;
				ErrorID := MC_ERROR_WRONG_MODE;
				state := 9999;
			ELSIF Ramp < 0 THEN
				Error := TRUE;
				ErrorID := MC_ERROR_PARAMETER_NOT_CORRECT;
				state := 9999;
//			ELSIF Backlash < -100 OR Backlash > 100 THEN
//				Error := TRUE;
//				ErrorID := MC_ERROR_PARAMETER_NOT_CORRECT;
//				state := 9999;
//			ELSIF Backlash = DEFAULT_BACKLASHVALUE THEN
//				(* read default backlash value *)
//				ReadParameter( Enable:= FALSE, Axis:= Axis);
//				Busy := TRUE;
//				state := 1;
			ELSIF Backlash = DEFAULT_BACKLASHVALUE THEN		(* HKP 2014-10-23 -  1) ersten auf diesen riesigen Defaultwert prüfen (1.0E307) *)
							(* read default backlash value *)
							ReadParameter( Enable:= FALSE, Axis:= Axis);
							Busy := TRUE;
							state := 1;
			ELSIF Backlash < -100 OR Backlash > 100 THEN	(* HKP 2014-10-23 -  2) erst dann auf sinnvolle User-Eingabe prüfen*)
							Error := TRUE;
							ErrorID := MC_ERROR_PARAMETER_NOT_CORRECT;
							state := 9999;
			ELSE
				iBacklash := Backlash;
				Busy := TRUE;
				state := 10;
			END_IF
		END_IF

	1: (* read default backlash value *)
		ReadParameter(
			Enable:= TRUE,
			ParameterNumber:= AxisBacklash,
			ReadMode:= READMODE_ONCE,
			Axis:= Axis );
		IF ReadParameter.Valid THEN
			iBacklash := ReadParameter.Value;
			IF iBacklash < -100 OR iBacklash > 100 THEN
				Error := TRUE;
				ErrorID := MC_ERROR_PARAMETER_NOT_CORRECT;
				state := 9999;
			ELSE
				state := 10;
			END_IF
		ELSIF ReadParameter.Error THEN
			Error := TRUE;
			ErrorID := ReadParameter.ErrorID;
			state := 9999;
		END_IF

	10 : (* active *)
		Enabled := TRUE;
		(*
		  1.)  Set backlash parameter in dependency of following input parameter: 'CompensationInPositiveDirection' (FALSE/TRUE)
			Remark: The sign of the 'Backlash' value (+/-) doesn't care.
		*)

		(* FALSE (default): backlash compensation must be done when driving in negative direction *)
		IF( NOT CompensationInPositiveDirection ) THEN
			stPosCompParameter.Direction		:= WorkDirectionNegative;
			stPosCompTable[0].Compensation	:= iBacklash;
			stPosCompTable[1].Compensation	:= iBacklash;
		(* TRUE: backlash compensation must be done when driving in positive direction *)
		ELSE
			stPosCompParameter.Direction		:= WorkDirectionPositive;
			stPosCompTable[0].Compensation	:= -iBacklash;
			stPosCompTable[1].Compensation	:= -iBacklash;
		END_IF

		(* BacklashValue = 0.0 *)
		IF ( iBacklash = 0.0 ) THEN
			stPosCompParameter.Direction		:= WorkDirectionNone;
			stPosCompTable[0].Compensation	:= 0.0;
			stPosCompTable[1].Compensation	:= 0.0;
		END_IF


		(* cycle time needed for pre calculation of the acceleration input *)
		IF CycleTime = 0 THEN
			GetThisTaskIndex();
			CycleTime := TwinCAT_SystemInfoVarList._TaskInfo[GetThisTaskIndex.index].cycleTime * LREAL#100E-9;
		END_IF

		(* special handling for disabling (depends from disable mode) *)
		IF( Enable = FALSE ) THEN
			(* disable mode HOLD *)
			IF( (DisableMode = DisableModeHold) ) THEN
				InternalEnable := TRUE;
				IF( Ramp > 0.0 ) THEN
					InternalAcceleration := Ramp / CycleTime;			(* mm/s^2 = mm/s / s *)
				ELSE
					InternalAcceleration := 0.0;
				END_IF
			(* disable mode RESET *)
			ELSE
				InternalEnable := Enable;
				InternalAcceleration := 0.0;
			END_IF
		(* active *)
		ELSE
			InternalEnable := Enable;
			IF( Ramp > 0.0 ) THEN
				InternalAcceleration := Ramp / CycleTime;				(* mm/s^2 = mm/s / s *)
			ELSE
				InternalAcceleration := 0.0;
			END_IF
		END_IF


		(* 2.) calculate backlash correction (if enabled) *)
		(* '_FB_PositionCorrectionTableLookup' *)
		fbCalcBacklashCorrection(
		   (* Enable := Enable, *)
		   Enable := InternalEnable,
		   pTable := ADR(stPosCompTable),
		   TableSize := SIZEOF(stPosCompTable),
		   Axis := Axis,
		   TableParameter := stPosCompParameter,
		   Compensation => InternalBacklashValue,
		   Error => CalcBacklashCorrOut.Error,
		   ErrorId => CalcBacklashCorrOut.ErrorID,
		   Active => CalcBacklashCorrOut.Active );

		(* check for error return code *)
		IF CalcBacklashCorrOut.Error THEN
			Error := TRUE;
			ErrorID := CalcBacklashCorrOut.ErrorID;
			state := 9999;
		END_IF


		(* 3.) feed backlash compensation (acceleration limited, that means linear velocity ramp) *)
		(*
				POSITIONCORRECTIONMODE_FAST
					The limitatation to maximum position change per cycle. Due to the maximum 
					change per cycle, the correction will take place as fast as possible and may 
					also be unlimited if PositionCorrectionValue is changed slightly. 
		*)
		(* MC_PositionCorrectionLimiter *)
		fbFeedBacklashCorrection(
		(*	Enable :=TRUE, *)
			 Enable :=Enable,
			 PositionCorrectionValue := InternalBacklashValue,
			 CorrectionMode := POSITIONCORRECTION_MODE_FAST,
		(*	 Acceleration := BacklashAccelecationLimit, *)	(* HKP: direct feeded user acceleration limit *)
			 Acceleration := InternalAcceleration,			(* HKP: pre calculated internal acceleration limit *)
			 CorrectionLength := 0.0,					(* optional length - not used for this correction mode 'POSITIONCORRECTION_MODE_FAST' *)
			 Axis := Axis,
			 Busy => FeedBacklashCorrOut.Busy,
			 Error => FeedBacklashCorrOut.Error,
			 ErrorID =>FeedBacklashCorrOut.ErrorID,
			 Limiting => InternalLimitingActive
			);

		(* check for error return code *)
		IF FeedBacklashCorrOut.Error THEN
			Error := TRUE;
			ErrorID := FeedBacklashCorrOut.ErrorID;
			state := 9999;
		END_IF


		CurrentBacklash	:= InternalBacklashValue;
		Limiting			:= InternalLimitingActive;

		IF NOT Enable THEN
			Enabled := FALSE;
			state := 0;
		END_IF

	9999 : (* error *)
		IF NOT Enable THEN
			Error := FALSE;
			ErrorID := 0;
			state := 0;
		END_IF
END_CASE

IF state = 0 THEN
	Busy := FALSE;
END_IF

END_FUNCTION_BLOCK

// POUs/Administrative/Extensions/MC_ReadDriveAddress
FUNCTION_BLOCK MC_ReadDriveAddress
(*	This Function Block returns the value of a vendor specific parameter *)
VAR_IN_OUT
	Axis				: AXIS_REF; (*Reference to an axis*)
END_VAR
VAR_INPUT
	Execute			: BOOL;
END_VAR
VAR_OUTPUT
	Done 			: BOOL;
	Busy			: BOOL;
	Error			: BOOL;
{attribute 'displaymode':='hex'}
	ErrorID			: UDINT;
	DriveAddress 	: ST_DriveAddress;
END_VAR
VAR
	state			: _E_TcMC_STATES := STATE_INITIALIZATION;
	TriggerExecute	: R_TRIG;
	fbAdsRead		: ADSREAD;
	readBuffer		: ARRAY[0..63] OF BYTE;	(* 2013-04-03 KSt - new data structure - size changed from 10 to 64 bytes *)
	
{attribute 'conditionalshow'}	i		: INT;
{attribute 'hide'}	pDword 	: POINTER TO DWORD;

	LastAxisId				: UDINT;
	LastControlLoopIndex	: UINT;
END_VAR

TriggerExecute(CLK:=Execute);

CASE state OF
	STATE_INITIALIZATION:
		IF NOT Execute THEN
			Done := FALSE;
			Error := FALSE;	(* reset at falling edge of Execute *)
			ErrorID := 0;
		END_IF
		IF TriggerExecute.Q THEN
			Done := FALSE;
			Busy := TRUE;
			Error := FALSE;
			ErrorID := 0;
			fbAdsRead(READ:=FALSE);
			(* read version of NC - 2013-04-03 KSt - read version dependent structure size *)
			(* 2017-11-10 skip when read drive address already done and AxisId and ControlLoopIndex has been unchanged *)
			IF Axis.DriveAddress.NetID <> ''
			  AND LastAxisId = Axis.NcToPlc.AxisId
			  AND LastControlLoopIndex = Axis.NcToPlc.ControlLoopIndex THEN
			  	LastAxisId := Axis.NcToPlc.AxisId;
				LastControlLoopIndex := Axis.NcToPlc.ControlLoopIndex;
				Done := TRUE;
				Busy := FALSE;
			ELSE	
				IF TcMcGlobal.NcDeviceInfoNcVersion=0 THEN
					TcMcGlobal.ReadDeviceInfo();
					state := STATE_WAITING;
				ELSE
					state := STATE_ORDER;
				END_IF
			END_IF
		END_IF

	STATE_WAITING : (* 2013-09-04 - new waiting state in case of invalid NC version information *)
		(* check for NC version *)
		TcMcGlobal.ReadDeviceInfo();
		IF NOT TcMcGlobal.fbADSRDDEVINFO.BUSY THEN
			state := STATE_ORDER;
		END_IF

	STATE_ORDER :
			IF TcMcGlobal.NcDeviceInfoNcVersion >= 16#03010FA2 (* Tc 3.1 NC4002 *) THEN
				fbAdsRead.LEN := SIZEOF(readBuffer);
			ELSIF TcMcGlobal.NcDeviceInfoNcVersion<16#03010000 AND TcMcGlobal.NcDeviceInfoNcVersion >= 16#03000BDB (* Tc 3.0 NC3035 *) THEN
				fbAdsRead.LEN := SIZEOF(readBuffer);
			ELSIF TcMcGlobal.NcDeviceInfoNcVersion<16#03000000 AND TcMcGlobal.NcDeviceInfoNcVersion >= 16#020B08B7 (* Tc 2.11 NC2231 *) THEN
				fbAdsRead.LEN := SIZEOF(readBuffer);
			ELSE
				MEMSET(ADR(readBuffer), SIZEOF(readBuffer), 0);
				fbAdsRead.LEN :=10; (* use old readbuffer size for compatibility reasons *)
			END_IF
			fbAdsRead(
				NETID:= TcMcGlobal.NCNETID_TCMC,
				PORT:= TcMcGlobal.NCPORT_TCMC,
				IDXGRP:=TcMcGlobal.Axis.Parameter.IDXGRP+Axis.NcToPlc.AxisId,
				IDXOFFS:= TcMcGlobal.Axis.Parameter.IDXOFFS.HWAMSADDR,
				LEN:= (* see above *),
				DESTADDR:= ADR(readBuffer),
				READ:= TRUE,
				TMOUT:= TcMcGlobal.tADSTimeOut );
			state := STATE_RUNNING;

	STATE_RUNNING:  (* wait until command is accepted *)
		fbAdsRead();
		IF NOT fbAdsRead.BUSY THEN
			Error := fbAdsRead.ERR;
			ErrorID := fbAdsRead.ERRID;
			IF NOT Error THEN
				FOR i := 0 TO 5 DO
					DriveAddress.NetIdBytes[i] := readBuffer[i];
				END_FOR
				DriveAddress.NetID := F_CreateAmsNetId( DriveAddress.NetIdBytes );
				DriveAddress.SlaveAddress := readBuffer[6] + 256* readBuffer[7];
				DriveAddress.Channel := readBuffer[8];
				pDword := ADR(readBuffer[12]);
				DriveAddress.NcDriveId := pDword^;
				pDword := ADR(readBuffer[16]);
				DriveAddress.NcDriveIndex := pDword^;
				pDword := ADR(readBuffer[20]);
				DriveAddress.NcDriveType := pDword^;
				pDword := ADR(readBuffer[24]);
				DriveAddress.NcEncoderId := pDword^;
				pDword := ADR(readBuffer[28]);
				DriveAddress.NcEncoderIndex := pDword^;
				pDword := ADR(readBuffer[32]);
				DriveAddress.NcEncoderType := pDword^;
				pDword := ADR(readBuffer[36]);
				DriveAddress.NcAxisId := pDword^;
				pDword := ADR(readBuffer[40]);
				DriveAddress.NcAxisType := pDword^;
				(* 2016-04-11 SoftDriveObjectId ab TcNc.sys 4226*)
				pDword := ADR(readBuffer[44]);
				DriveAddress.TcSoftDriveObjectId := pDword^;
				DriveAddress.TcDriveObjectId := pDword^;
				(* 2018-06-06 SoftDriveObjectId ab TcNc.sys xxxx*)
				pDword := ADR(readBuffer[48]);
				DriveAddress.TcEncoderObjectId := pDword^;
				
				DriveAddress.TcAxisObjectId := _F_GetTcAxisObjectId(AxisId := Axis.NcToPlc.AxisId);
				
				Axis.DriveAddress := DriveAddress;

			  	LastAxisId := Axis.NcToPlc.AxisId;
				LastControlLoopIndex := Axis.NcToPlc.ControlLoopIndex;
			END_IF
			Done := NOT Error;
			Busy := FALSE;
			fbAdsRead(READ:=FALSE);
			state := STATE_INITIALIZATION;  (* wait until command is accepted *)
		END_IF
END_CASE

END_FUNCTION_BLOCK

// POUs/Administrative/Extensions/MC_SetAcceptBlockedDriveSignal
FUNCTION MC_SetAcceptBlockedDriveSignal : BOOL
(* 	reference: 	PLC -> NC axis interface (128 bytes)
	copy the signal to bit 8 of an axis nDeCtrlDWord:

	- Accept blocked drive (accept that drive does not follow the controllers
	set point values - e. g. when homing on the limit switches)

	- Akzeptiere blockierten Antrieb (akzeptiere, dass der Antrieb den  
 	Sollwerten nicht folgt - z. B. beim Referenzieren auf Endschalter)
*)
VAR_IN_OUT
	Axis				: AXIS_REF; (*Reference to an axis*)
END_VAR
VAR_INPUT
	Enable : BOOL;
END_VAR
VAR
END_VAR

Axis.PlcToNc.ControlDWord.8 := Enable;
MC_SetAcceptBlockedDriveSignal := Enable;

END_FUNCTION

// POUs/Administrative/Status and Parameter/MC_WriteBoolParameterPersistent
FUNCTION_BLOCK MC_WriteBoolParameterPersistent
VAR_IN_OUT
	Axis: AXIS_REF; (*Reference to an axis*)
END_VAR
VAR_INPUT
	Execute: BOOL;
	ParameterNumber: MC_AxisParameter; // 2023-03 KSt changed from INT to MC_AxisParameter
	Value: BOOL;
END_VAR
VAR_OUTPUT
	Done: BOOL;
	Busy: BOOL;
	Error: BOOL;
{attribute 'displaymode':='hex'}
	ErrorID: UDINT;
END_VAR
VAR
	fbWriteParameterPersistent: _FB_WriteParameterPersistent;
END_VAR

fbWriteParameterPersistent(
	Axis:= Axis, 
	Execute:= Execute, 
	ParameterNumber:= ParameterNumber, 
	Value:= SEL(Value, 0, 1), 
//	ParameterType:= PARAMETERTYPE_BOOL, 	(* removed 2018-11-22 KSt - not required *)
	Done=> Done, 
	Busy=> Busy, 
	Error=> Error, 
	ErrorID=> ErrorID);

END_FUNCTION_BLOCK

// POUs/Administrative/Extensions/DriveOperationMode/MC_ReadDriveOperationMode
{attribute 'conditionalshow_all_locals'}
FUNCTION_BLOCK MC_ReadDriveOperationMode 
(*	This function block returns the current drive operation mode
*)
VAR_IN_OUT
	Axis			:	AXIS_REF; (*Reference to an axis*)
END_VAR
VAR_INPUT
	Execute			:	BOOL;	(* B *)
	Options			: ST_DriveOperationModeOptions;
END_VAR
VAR_OUTPUT
	Done 			: 	BOOL;	(* B *)
	Busy			: 	BOOL;	(* E *)
	Error 			: 	BOOL;	(* B *)
{attribute 'displaymode':='hex'}
	ErrorID 		: 	UDINT;	(* E *)
	DriveOperationMode 	: 	E_DriveOperationMode;
END_VAR
VAR
	TriggerExecute: R_TRIG;
	state: _E_TcMC_STATES := STATE_INITIALIZATION;
	stReadDriveOperationModeRequest : _ST_TcNC_ReadDriveOperationModeRequest;
	stReadDriveOperationModeResponse : _ST_TcNC_ReadDriveOperationModeResponse;
	fbAdsReadWrite		: 	ADSRDWRT;
END_VAR

TriggerExecute(CLK:=Execute);

CASE state OF
	STATE_INITIALIZATION:
		IF NOT Execute THEN
			Done := FALSE;
			Error := FALSE;	(* reset at falling edge of Execute *)
			ErrorID := 0;
		END_IF
		IF TriggerExecute.Q THEN
			Done := FALSE;
			Busy := TRUE;
			Error := FALSE;
			ErrorID := 0;
			DriveOperationMode := 0 ;
			stReadDriveOperationModeRequest.nReserved1 := 0;
			stReadDriveOperationModeRequest.nReserved2 := 0;
			fbAdsReadWrite(WRTRD:=FALSE);
		END_IF
		IF Busy THEN
			fbAdsReadWrite(
				NETID:= TcMcGlobal.NCNETID_TCMC,
				PORT:= AMSPORT_R0_NCSAF,
				IDXGRP:=TcMcGlobal.Axis.State.IDXGRP+Axis.NcToPlc.AxisId,
				IDXOFFS:= 16#63, //TcMcGlobal.Axis.State.IDXOFFS.STOPINFORMATION,
				WRITELEN:= SIZEOF(stReadDriveOperationModeRequest),
				READLEN:= SIZEOF(stReadDriveOperationModeResponse),
				SRCADDR:= ADR(stReadDriveOperationModeRequest),
				DESTADDR:= ADR(stReadDriveOperationModeResponse),
				WRTRD:= TRUE,
				TMOUT:= TcMcGlobal.tADSTimeOut );
			IF NOT fbAdsReadWrite.BUSY THEN
				Error := fbAdsReadWrite.ERR;
				ErrorID := fbAdsReadWrite.ERRID;
				Done := NOT Error;
				IF Done THEN
					DriveOperationMode := stReadDriveOperationModeResponse.eTcNc3DrvOpMode;
				END_IF
				Busy := FALSE;
			END_IF
		END_IF
END_CASE

END_FUNCTION_BLOCK

// POUs/Administrative/Extensions/DriveOperationMode/MC_WriteDriveOperationMode
{attribute 'conditionalshow_all_locals'}
FUNCTION_BLOCK MC_WriteDriveOperationMode 
VAR_IN_OUT
	Axis : AXIS_REF; (*Reference to an axis*)
END_VAR
VAR_INPUT
	Execute : BOOL;
	DriveOperationMode : E_DriveOperationMode;
	Options	: ST_DriveOperationModeOptions;
END_VAR
VAR_OUTPUT
	Done : BOOL;
	Busy : BOOL;
	Error : BOOL;
{attribute 'displaymode':='hex'}
	ErrorID : UDINT;
END_VAR
VAR
	LastExecutionResult: 	_ST_FunctionBlockResults;
	ADSbusy: BOOL;
	state: _E_TcMC_STATES := STATE_INITIALIZATION;
	stWriteDriveOperationMode : _ST_TcNC_WriteDriveOperationMode;
	fbADSWRITE: ADSWRITE;
END_VAR
VAR
	TriggerExecute: R_TRIG;
END_VAR

TriggerExecute(CLK:=Execute);

CASE state OF
	STATE_INITIALIZATION :
		Busy := FALSE;
		IF NOT Execute THEN
			Done := FALSE;
			Error := FALSE;
			ErrorID := 0;
		END_IF
		IF TriggerExecute.Q THEN		
			Busy := TRUE;

			LastExecutionResult.Done := FALSE;
			LastExecutionResult.CommandAborted := FALSE;
			LastExecutionResult.Error := FALSE;
			LastExecutionResult.ErrorID := 0;
	
			IF DriveOperationMode <> E_DriveOperationMode.DriveOperationMode_Default
			  AND DriveOperationMode <> E_DriveOperationMode.DriveOperationMode_Torque
			  AND DriveOperationMode <> E_DriveOperationMode.DriveOperationMode_Velo1
			  AND DriveOperationMode <> E_DriveOperationMode.DriveOperationMode_Velo2
			  AND DriveOperationMode <> E_DriveOperationMode.DriveOperationMode_Pos1
			  AND DriveOperationMode <> E_DriveOperationMode.DriveOperationMode_Pos2
			  AND DriveOperationMode <> E_DriveOperationMode.DriveOperationMode_TorqueAndCommutationAngle
			  AND DriveOperationMode <> E_DriveOperationMode.DriveOperationMode_VelocityMode
			  AND DriveOperationMode <> E_DriveOperationMode.DriveOperationMode_DriveBasedHoming
			  AND DriveOperationMode <> E_DriveOperationMode.DriveOperationMode_Index0
			  AND DriveOperationMode <> E_DriveOperationMode.DriveOperationMode_Index1
			  AND DriveOperationMode <> E_DriveOperationMode.DriveOperationMode_Index2
			  AND DriveOperationMode <> E_DriveOperationMode.DriveOperationMode_Index3
			  AND DriveOperationMode > 0 THEN  
				Busy := FALSE;
				Error := TRUE;
				ErrorID := MC_ERROR_WRONG_MODE;
			ELSE
				stWriteDriveOperationMode.eTcNc3DrvOpMode := DriveOperationMode;
				stWriteDriveOperationMode.nReserved0 := 0;
				stWriteDriveOperationMode.nReserved1 := 0;
				stWriteDriveOperationMode.nReserved2 := 0;
				
